// SIMATIC STEP 7 (V5.x) project Ciclo ppal
// program: Programa S7(2)
// program: TEST_DESBOBINADO
// program: TEST_CIZALLADO
// program: TEST_M_DESBOBINADO
// program: TEST_M_CIZALLADO
// program: TEST_G_DESBOBINADO
// program: TEST_G_CIZALLADO
// program: TEST_MODOS
// program: TEST_PESAJE
// program: TEST_GENERAL
// program: TEST_CORTAR
// program: TEST_ERRORES

SYMBOL_TABLE
"CONTADOR"	C 1	COUNTER	// Cuenta el numero de planchas cortadas
"Global"	DB 1	DB 1
"Modo1"	DB 2	DB 2
"Modo2"	DB 3	DB 3
"INFO_BOB"	DB 4	DB 4
"DESBOBINADO"	FB 1	FB 1	// Función que se encarga del desbobinado
"CIZALLADO"	FB 2	FB 2	// Funcion que se encaga del cizallado de planchas
"MULT_DESBOB"	FB 3	FB 3
"MULT_CIZA"	FB 4	FB 4
"GENERAL"	FB 5	FB 5
"MULT_GEN_DESB"	FB 6	FB 6
"MULT_GEN_CIZA"	FB 7	FB 7
"CORTA"	FB 8	FB 8
"MODO"	FB 9	FB 9
"ERRORES"	FC 1	FC 1
"PESAJE"	FC 2	FC 2	// Función de pesaje
"SCALE"	FC 105	FC 105	// Scaling Values
"BOBINA_COLOCADA"	I 124.0	BOOL
"S_SARTEN"	I 124.1	BOOL
"S_CACEROLA"	I 124.2	BOOL
"S_WOK"	I 124.3	BOOL
"S_PAELLERA"	I 124.4	BOOL
"PRESENCIA"	I 124.5	BOOL
"PALET"	I 124.6	BOOL
"SENSORARRIBA"	I 124.7	BOOL
"SENSORABAJO"	I 125.0	BOOL
"EXPULSADA"	I 125.1	BOOL
"ON"	I 125.2	BOOL
"BDT"	I 125.3	BOOL
"MODO_1"	I 125.4	BOOL
"MODO_2"	I 125.5	BOOL
"RESET"	I 125.6	BOOL
"SETA_PELIGROSA"	I 125.7	BOOL
"ERROR"	M 124.0	BOOL
"PESO_OUT"	MD 300	REAL
"CYCL_EXC"	OB 1	OB 1	// Cycle Execution
"MCENTRO"	PIW 651	INT
"IN_PESAJE"	PIW 653	INT
"ABRIRMCENTRO"	Q 100.0	BOOL
"CERRARMCENTRO"	Q 100.1	BOOL
"DESBOBINAR"	Q 100.2	BOOL
"EXPULSAR_BOBINA"	Q 100.3	BOOL
"EXPULSAR_PLANCHA"	Q 100.4	BOOL
"BAJAR_CUCHILLA"	Q 100.5	BOOL
"EXPULSAR_PALET"	Q 100.6	BOOL
"PRENSA"	Q 100.7	BOOL
"STBY_DESBOB"	Q 101.0	BOOL
"STBY_CIZA"	Q 101.1	BOOL
"TEMP_ERROR"	T 1	TIMER
END_SYMBOL_TABLE

FUNCTION_BLOCK "DESBOBINADO"	// FB 1
TITLE = DESBOBINADO
VERSION : 0.1
VAR_INPUT
  SENSOR : BOOL ;
  PRESENCIA : BOOL ;
  CENTRO : INT ;
  MCENTRO : INT ;
  Contador : COUNTER ;
  START : BOOL ;
  PLANCHAS : WORD  := W#16#100;
  ERROR : BOOL ;
  RESET : BOOL ;
END_VAR
VAR_OUTPUT
  ABRIRMCENTRO : BOOL ;
  DESBOBINAR : BOOL ;
  STBY : BOOL ;
END_VAR
VAR
  x31 : BOOL ;
  x32 : BOOL ;
  x33 : BOOL ;
  x34 : BOOL ;
  x30 : BOOL ;
  FP_PRESENCIA : BOOL ;
  BDT : BOOL ;
  FP_START : BOOL ;
  XERROR : BOOL ;
END_VAR
VAR_TEMP
  watchdog_master : BOOL ;
END_VAR
BEGIN
NETWORK
TITLE = Arranque
      SET;
      FP    #BDT;
      S     #x30;
      R     #x31;
      R     #x32;
      R     #x33;
      R     #x34;
NETWORK
TITLE =
      A     #RESET;
      R     #ABRIRMCENTRO;
      R     #DESBOBINAR;
      S     #x30;
      R     #x31;
      R     #x32;
      R     #x33;
      R     #x34;
      R     #XERROR;
NETWORK
TITLE =
      A     #ERROR;
      R     #ABRIRMCENTRO;
      R     #DESBOBINAR;
      R     #x30;
      R     #x31;
      R     #x32;
      R     #x33;
      R     #x34;
      S     #XERROR;
NETWORK
TITLE = x31 a x32
//Comparacion medida centro con medida nominal del centro para pasar de x31 a x32
      A     #x31;
      A(;
      L     #CENTRO;
      L     #MCENTRO;
      ==R;
      );
      R     #x31;
      S     #x32;
NETWORK
TITLE = x32 a x33
//Presencia detecta que la plancha esta en posicion para empezar el proceso de 
//desbobinado-cizallado
      A     #x32;
      A     #PRESENCIA;
      FP    #FP_PRESENCIA;
      R     #x32;
      S     #x33;
NETWORK
TITLE = x33 a x34
//Detecta que la plancha esta lista para ser cizallada
      A     #x33;
      A     #SENSOR;
      R     #x33;
      S     #x34;
NETWORK
TITLE = x34 a x33
//si el contador no ha acabado
      A     #x34;
      T     LD 1;
      TAK;
      T     LD 5;
      L     #Contador;
      T     LW 9;
      L     LD 5;
      L     LD 1;
      A     C [LW 9];
      AN    #SENSOR;
      R     #x34;
      S     #x33;
NETWORK
TITLE = x34 a X30
//si el contador ha cabado
      A     #x34;
      T     LD 1;
      TAK;
      T     LD 5;
      L     #Contador;
      T     LW 9;
      L     LD 5;
      L     LD 1;
      AN    C [LW 9];
      AN    #SENSOR;
      AN    #PRESENCIA;
      R     #x34;
      S     #x30;
NETWORK
TITLE = Tratamiento de bit de fin
      A     #x30;
      =     #STBY;
NETWORK
TITLE = Abrir centro
      A     #x31;
      =     #ABRIRMCENTRO;
NETWORK
TITLE = Carga del contador y desbobinado en x32
      A     #x32;
      S     #DESBOBINAR;
      L     #PLANCHAS;
      T     LD 1;
      TAK;
      T     LD 5;
      L     #Contador;
      T     LW 9;
      L     LD 5;
      L     LD 1;
      S     C [LW 9];
NETWORK
TITLE = Resta del contador y salida del x33
      A     #x33;
      S     #DESBOBINAR;
NETWORK
TITLE = Reset del desbobionado en x34
      A     #x34;
      R     #DESBOBINAR;
NETWORK
TITLE = De X30 a X31
      A     #START;
      FP    #FP_START;
      A     #x30;
      R     #x30;
      S     #x31;
END_FUNCTION_BLOCK

FUNCTION_BLOCK "CIZALLADO"	// FB 2
TITLE = CIZALLADO
VERSION : 0.1
VAR_INPUT
  SENSOR : BOOL ;
  SENSORABAJO : BOOL ;
  SENSORARRIBA : BOOL ;
  EXPULSADA : BOOL ;
  CONTADOR : COUNTER ;
  START : BOOL ;
  RESET : BOOL ;
  ERROR : BOOL ;
END_VAR
VAR_OUTPUT
  BAJARCUCHILLA : BOOL ;
  EXPULSARPLANCHA : BOOL ;
  STBY : BOOL ;
  BIT_OK : BOOL ;
END_VAR
VAR
  X41 : BOOL ;
  M3 : BOOL ;
  X43 : BOOL ;
  BDT : BOOL ;
  FP_START : BOOL ;
  INICORTAR : BOOL ;
  S2 : BOOL ;
  OK_CORTAR : BOOL ;
  STBY_CORTAR : BOOL ;
  CORTADO : BOOL ;
  XERROR : BOOL ;
  CORTAR : FB 8;
END_VAR
BEGIN
NETWORK
TITLE = Arranque
      SET;
      FP    #BDT;
      S     #X41;
      R     #M3;
      R     #X43;
      R     #INICORTAR;
      R     #CORTADO;
      R     #BIT_OK;
      R     #S2;
NETWORK
TITLE = De x41 a M3
      A     #X41;
      A     #SENSOR;
      A     #STBY_CORTAR;
      A     #START;
      FP    #FP_START;
      R     #X41;
      S     #M3;
NETWORK
TITLE = De M3 a x43
      A     #M3;
      A     #CORTADO;
      R     #M3;
      S     #X43;
NETWORK
TITLE = de x43 a x41
      A     #X43;
      A     #STBY_CORTAR;
      T     LD 0;
      TAK;
      T     LD 4;
      L     #CONTADOR;
      T     LW 8;
      L     LD 4;
      L     LD 0;
      AN    C [LW 8];
      R     #X43;
      S     #S2;
NETWORK
TITLE = de x43 a X41
      A     #X43;
      A     #STBY_CORTAR;
      T     LD 0;
      TAK;
      T     LD 4;
      L     #CONTADOR;
      T     LW 8;
      L     LD 4;
      L     LD 0;
      A     C [LW 8];
      R     #X43;
      S     #X41;
NETWORK
TITLE = Call M3
      CALL  #CORTAR (
           SENSORABAJO              := #SENSORABAJO,
           SENSORARRIBA             := #SENSORARRIBA,
           EXPULSADA                := #EXPULSADA,
           START                    := #INICORTAR,
           OK                       := #OK_CORTAR,
           ERROR                    := #ERROR,
           RESET                    := #RESET,
           BAJARCUCHILLA            := #BAJARCUCHILLA,
           EXPULSARPLANCHA          := #EXPULSARPLANCHA,
           BIT_OK                   := #CORTADO,
           STBY                     := #STBY_CORTAR);
NETWORK
TITLE = De M3 a X43
      A     #M3;
      A     #CORTADO;
      R     #M3;
      S     #X43;
NETWORK
TITLE = Salida M3
      A     #M3;
      =     #INICORTAR;
NETWORK
TITLE = Cuenta el numero de planchas cortadas
      A     #X43;
      =     #OK_CORTAR;
      T     LD 0;
      TAK;
      T     LD 4;
      L     #CONTADOR;
      T     LW 8;
      L     LD 4;
      L     LD 0;
      CD    C [LW 8];
NETWORK
TITLE = Salida X41
      A     #X41;
      =     #STBY;
NETWORK
TITLE = Salida S2
      A     #S2;
      =     #BIT_OK;
NETWORK
TITLE =
      A     #RESET;
      S     #X41;
      R     #M3;
      R     #X43;
      R     #INICORTAR;
      R     #CORTADO;
      R     #BIT_OK;
      R     #S2;
      R     #XERROR;
NETWORK
TITLE =
      A     #ERROR;
      R     #X41;
      R     #M3;
      R     #X43;
      R     #INICORTAR;
      R     #CORTADO;
      R     #BIT_OK;
      R     #S2;
      S     #XERROR;
END_FUNCTION_BLOCK

FUNCTION_BLOCK "MULT_DESBOB"	// FB 3
VERSION : 0.1
VAR_INPUT
  S_CACEROLA : BOOL ;
  S_SARTEN : BOOL ;
  S_PAELLERA : BOOL ;
  S_WOK : BOOL ;
  PRESENCIA : BOOL ;
  C_CACEROLA : INT ;
  C_SARTEN : INT ;
  C_WOK : INT ;
  C_PAELLERA : INT ;
  MCENTRO : INT ;
  CONTADOR : COUNTER ;
  PLANCHAS : WORD ;
  SARTEN : BOOL ;
  CACEROLA : BOOL ;
  WOK : BOOL ;
  PAELLERA : BOOL ;
  START : BOOL ;
  ERROR : BOOL ;
  RESET : BOOL ;
END_VAR
VAR_OUTPUT
  ABRIRMCENTRO : BOOL ;
  DESBOBINAR : BOOL ;
  BIT_OK : BOOL ;
  BIT_ERROR : BOOL ;
  STBY : BOOL ;
  STBY_SAR : BOOL ;
  STBY_CAC : BOOL ;
  STBY_WOK : BOOL ;
  STBY_PAELL : BOOL ;
END_VAR
VAR
  START_SAR : BOOL ;
  START_CAC : BOOL ;
  START_WOK : BOOL ;
  START_PAELL : BOOL ;
  FP_BDT : BOOL ;
  X1 : BOOL ;
  X2 : BOOL ;
  X3 : BOOL ;
  X4 : BOOL ;
  X5 : BOOL ;
  X6 : BOOL ;
  BDT : BOOL ;
  FP_START : BOOL ;
  FLAG_DESB : BOOL ;
  FP_DESBOB : BOOL ;
  F_START : BOOL ;
  FN_BDT : BOOL ;
  FN_X1 : BOOL ;
  SAR_DESBOB : FB 1;
  CAC_DESBOB : FB 1;
  WOK_DESBOB : FB 1;
  PAELL_DESBOB : FB 1;
END_VAR
BEGIN
NETWORK
TITLE = call del x2
      A     #X2;
      JCN   _001;
      S     #BDT;
      BLD   14;
      =     L 6.0;
      L     DINO;
      T     LW 4;
      CDB;
      OPN   DI [LW 4];
      TAR2  LD 0;
      A     DBX [AR2,P#0.1];
      =     #SAR_DESBOB.SENSOR;
      A     DBX [AR2,P#0.4];
      =     #SAR_DESBOB.PRESENCIA;
      L     DBW [AR2,P#4.0];
      T     #SAR_DESBOB.CENTRO;
      L     DBW [AR2,P#10.0];
      T     #SAR_DESBOB.MCENTRO;
      L     DBW [AR2,P#12.0];
      T     #SAR_DESBOB.Contador;
      A     DBX [AR2,P#20.0];
      =     #SAR_DESBOB.START;
      L     DBW [AR2,P#14.0];
      T     #SAR_DESBOB.PLANCHAS;
      A     DBX [AR2,P#16.5];
      =     #SAR_DESBOB.ERROR;
      A     DBX [AR2,P#16.6];
      =     #SAR_DESBOB.RESET;
      +AR2  P#24.0;
      UC    "DESBOBINADO";
      LAR2  LD 0;
      A     #SAR_DESBOB.ABRIRMCENTRO;
      =     DBX [AR2,P#18.0];
      A     #SAR_DESBOB.DESBOBINAR;
      =     DBX [AR2,P#18.1];
      A     #SAR_DESBOB.STBY;
      =     DBX [AR2,P#18.5];
      CDB;
      BLD   15;
_001: NOP   0;
NETWORK
TITLE = call del x3
      A     #X3;
      JCN   _002;
      S     #BDT;
      BLD   14;
      =     L 6.0;
      L     DINO;
      T     LW 4;
      CDB;
      OPN   DI [LW 4];
      TAR2  LD 0;
      A     DBX [AR2,P#0.0];
      =     #CAC_DESBOB.SENSOR;
      A     DBX [AR2,P#0.4];
      =     #CAC_DESBOB.PRESENCIA;
      L     DBW [AR2,P#2.0];
      T     #CAC_DESBOB.CENTRO;
      L     DBW [AR2,P#10.0];
      T     #CAC_DESBOB.MCENTRO;
      L     DBW [AR2,P#12.0];
      T     #CAC_DESBOB.Contador;
      A     DBX [AR2,P#20.1];
      =     #CAC_DESBOB.START;
      L     DBW [AR2,P#14.0];
      T     #CAC_DESBOB.PLANCHAS;
      A     DBX [AR2,P#16.5];
      =     #CAC_DESBOB.ERROR;
      A     DBX [AR2,P#16.6];
      =     #CAC_DESBOB.RESET;
      +AR2  P#42.0;
      UC    "DESBOBINADO";
      LAR2  LD 0;
      A     #CAC_DESBOB.ABRIRMCENTRO;
      =     DBX [AR2,P#18.0];
      A     #CAC_DESBOB.DESBOBINAR;
      =     DBX [AR2,P#18.1];
      A     #CAC_DESBOB.STBY;
      =     DBX [AR2,P#18.6];
      CDB;
      BLD   15;
_002: NOP   0;
NETWORK
TITLE = call del x4
      A     #X4;
      JCN   _003;
      S     #BDT;
      BLD   14;
      =     L 6.0;
      L     DINO;
      T     LW 4;
      CDB;
      OPN   DI [LW 4];
      TAR2  LD 0;
      A     DBX [AR2,P#0.3];
      =     #WOK_DESBOB.SENSOR;
      A     DBX [AR2,P#0.4];
      =     #WOK_DESBOB.PRESENCIA;
      L     DBW [AR2,P#6.0];
      T     #WOK_DESBOB.CENTRO;
      L     DBW [AR2,P#10.0];
      T     #WOK_DESBOB.MCENTRO;
      L     DBW [AR2,P#12.0];
      T     #WOK_DESBOB.Contador;
      A     DBX [AR2,P#20.2];
      =     #WOK_DESBOB.START;
      L     DBW [AR2,P#14.0];
      T     #WOK_DESBOB.PLANCHAS;
      A     DBX [AR2,P#16.5];
      =     #WOK_DESBOB.ERROR;
      A     DBX [AR2,P#16.6];
      =     #WOK_DESBOB.RESET;
      +AR2  P#60.0;
      UC    "DESBOBINADO";
      LAR2  LD 0;
      A     #WOK_DESBOB.ABRIRMCENTRO;
      =     DBX [AR2,P#18.0];
      A     #WOK_DESBOB.DESBOBINAR;
      =     DBX [AR2,P#18.1];
      A     #WOK_DESBOB.STBY;
      =     DBX [AR2,P#18.7];
      CDB;
      BLD   15;
_003: NOP   0;
NETWORK
TITLE = call del x5
      A     #X5;
      JCN   _004;
      S     #BDT;
      BLD   14;
      =     L 6.0;
      L     DINO;
      T     LW 4;
      CDB;
      OPN   DI [LW 4];
      TAR2  LD 0;
      A     DBX [AR2,P#0.2];
      =     #PAELL_DESBOB.SENSOR;
      A     DBX [AR2,P#0.4];
      =     #PAELL_DESBOB.PRESENCIA;
      L     DBW [AR2,P#8.0];
      T     #PAELL_DESBOB.CENTRO;
      L     DBW [AR2,P#10.0];
      T     #PAELL_DESBOB.MCENTRO;
      L     DBW [AR2,P#12.0];
      T     #PAELL_DESBOB.Contador;
      A     DBX [AR2,P#20.3];
      =     #PAELL_DESBOB.START;
      L     DBW [AR2,P#14.0];
      T     #PAELL_DESBOB.PLANCHAS;
      A     DBX [AR2,P#16.5];
      =     #PAELL_DESBOB.ERROR;
      A     DBX [AR2,P#16.6];
      =     #PAELL_DESBOB.RESET;
      +AR2  P#78.0;
      UC    "DESBOBINADO";
      LAR2  LD 0;
      A     #PAELL_DESBOB.ABRIRMCENTRO;
      =     DBX [AR2,P#18.0];
      A     #PAELL_DESBOB.DESBOBINAR;
      =     DBX [AR2,P#18.1];
      A     #PAELL_DESBOB.STBY;
      =     DBX [AR2,P#18.4];
      CDB;
      BLD   15;
_004: NOP   0;
NETWORK
TITLE = salida x2
      A     #X2;
      =     #START_SAR;
NETWORK
TITLE = salida x3
      A     #X3;
      =     #START_CAC;
NETWORK
TITLE = salida x4
      A     #X4;
      =     #START_WOK;
NETWORK
TITLE = salida x5
      A     #X5;
      =     #START_PAELL;
NETWORK
TITLE = Arranque
      SET;
      FP    #FP_BDT;
      R     #START_SAR;
      R     #START_CAC;
      R     #START_WOK;
      R     #START_PAELL;
      S     #X1;
      R     #X2;
      R     #X3;
      R     #X4;
      R     #X5;
      R     #X6;
NETWORK
TITLE = guardado de flanco de start
      A     #START;
      FP    #FP_START;
      =     #F_START;
NETWORK
TITLE = de x1 x2
      A     #F_START;
      A     #X1;
      A     #SARTEN;
      R     #X1;
      S     #X2;
NETWORK
TITLE = de x1 a x3
      A     #F_START;
      A     #X1;
      A     #CACEROLA;
      R     #X1;
      S     #X3;
NETWORK
TITLE = de x1 a x4
      A     #F_START;
      A     #X1;
      A     #WOK;
      R     #X1;
      S     #X4;
NETWORK
TITLE = de x1 a x5
      A     #F_START;
      A     #X1;
      A     #PAELLERA;
      R     #X1;
      S     #X5;
NETWORK
TITLE = Guardado flag desbobinado
      A     #DESBOBINAR;
      FP    #FP_DESBOB;
      S     #FLAG_DESB;
NETWORK
TITLE = de x2 a x6
      A     #X2;
      A     #FLAG_DESB;
      A     #STBY_SAR;
      R     #FLAG_DESB;
      R     #X2;
      S     #X6;
NETWORK
TITLE = de x3 a x6
      A     #X3;
      A     #FLAG_DESB;
      A     #STBY_CAC;
      R     #FLAG_DESB;
      R     #X3;
      S     #X6;
NETWORK
TITLE = de x4 a x6
      A     #X4;
      A     #FLAG_DESB;
      A     #STBY_WOK;
      R     #FLAG_DESB;
      R     #X4;
      S     #X6;
NETWORK
TITLE = de x5 a x6
      A     #X5;
      A     #FLAG_DESB;
      A     #STBY_PAELL;
      R     #FLAG_DESB;
      R     #X5;
      S     #X6;
NETWORK
TITLE = salida x1
      A     #X1;
      =     #STBY;
NETWORK
TITLE = salida x6 
      A     #X6;
      =     #BIT_OK;
NETWORK
TITLE = error, sin prgramar
      A     #RESET;
      A(;
      A(;
      O(;
      A     #STBY_CAC;
      A     #X3;
      );
      O(;
      A     #STBY_SAR;
      A     #X2;
      );
      O(;
      A     #STBY_WOK;
      A     #X4;
      );
      O(;
      A     #STBY_PAELL;
      A     #X5;
      );
      );
      O     #X6;
      );
      R     #BDT;
      R     #BIT_OK;
      R     #BIT_ERROR;
      S     #X1;
      R     #X2;
      R     #X3;
      R     #X4;
      R     #X5;
      R     #X6;
      R     #START_SAR;
      R     #START_CAC;
      R     #START_WOK;
      R     #START_PAELL;
      R     #FLAG_DESB;
      R     #ABRIRMCENTRO;
      R     #DESBOBINAR;
END_FUNCTION_BLOCK

FUNCTION_BLOCK "MULT_CIZA"	// FB 4
VERSION : 0.1
VAR_INPUT
  S_CACEROLA : BOOL ;
  S_WOK : BOOL ;
  S_SARTEN : BOOL ;
  S_PAELLERA : BOOL ;
  SENSORARRIBA : BOOL ;
  SENSORABAJO : BOOL ;
  EXPULSADA : BOOL ;
  CONTADOR : COUNTER ;
  SARTEN : BOOL ;
  CACEROLA : BOOL ;
  WOK : BOOL ;
  PAELLERA : BOOL ;
  START : BOOL ;
  ERROR : BOOL ;
  RESET : BOOL ;
END_VAR
VAR_OUTPUT
  EXPULSARPLANCHA : BOOL ;
  BAJARCUCHILLA : BOOL ;
  BIT_OK : BOOL ;
  STBY : BOOL ;
END_VAR
VAR
  START_SAR : BOOL ;
  START_CAC : BOOL ;
  START_WOK : BOOL ;
  START_PAELL : BOOL ;
  X1 : BOOL ;
  X2 : BOOL ;
  X3 : BOOL ;
  X4 : BOOL ;
  X5 : BOOL ;
  FP_START : BOOL ;
  F_START : BOOL ;
  STBY_SAR : BOOL ;
  STBY_CAC : BOOL ;
  STBY_WOK : BOOL ;
  STBY_PAELL : BOOL ;
  OK : BOOL ;
  BDT : BOOL ;
  X6 : BOOL ;
  RESET_CIZA : BOOL ;
  FP_RESET : BOOL ;
  CAC_CIZA : FB 2;
  SAR_CIZA : FB 2;
  WOK_CIZA : FB 2;
  PAELL_CIZA : FB 2;
END_VAR
BEGIN
NETWORK
TITLE = Arranque
      SET;
      FP    #BDT;
      S     #X1;
      R     #X2;
      R     #X3;
      R     #X4;
      R     #X5;
      R     #X6;
NETWORK
TITLE = De x1 a x2
      A     #START;
      A     #SARTEN;
      A     #X1;
      R     #X1;
      S     #X2;
NETWORK
TITLE = de x1 a x3
      A     #START;
      A     #CACEROLA;
      A     #X1;
      R     #X1;
      S     #X3;
NETWORK
TITLE = de x1 a x4
      A     #START;
      A     #WOK;
      A     #X1;
      R     #X1;
      S     #X4;
NETWORK
TITLE = de x1 a x5
      A     #START;
      A     #PAELLERA;
      A     #X1;
      R     #X1;
      S     #X5;
NETWORK
TITLE = de x2-5 a x1
      A     #OK;
      A(;
      O     #X2;
      O     #X3;
      O     #X4;
      O     #X5;
      );
      R     #X2;
      R     #X3;
      R     #X4;
      R     #X5;
      S     #X1;
NETWORK
TITLE = call del x2
      A     #X2;
      JCN   _001;
      BLD   14;
      =     L 6.0;
      L     DINO;
      T     LW 4;
      CDB;
      OPN   DI [LW 4];
      TAR2  LD 0;
      A     DBX [AR2,P#0.2];
      =     #SAR_CIZA.SENSOR;
      A     DBX [AR2,P#0.5];
      =     #SAR_CIZA.SENSORABAJO;
      A     DBX [AR2,P#0.4];
      =     #SAR_CIZA.SENSORARRIBA;
      A     DBX [AR2,P#0.6];
      =     #SAR_CIZA.EXPULSADA;
      L     DBW [AR2,P#2.0];
      T     #SAR_CIZA.CONTADOR;
      A     DBX [AR2,P#8.0];
      =     #SAR_CIZA.START;
      A     DBX [AR2,P#10.2];
      =     #SAR_CIZA.RESET;
      A     DBX [AR2,P#4.5];
      =     #SAR_CIZA.ERROR;
      +AR2  P#28.0;
      UC    "CIZALLADO";
      LAR2  LD 0;
      A     #SAR_CIZA.BAJARCUCHILLA;
      =     DBX [AR2,P#6.1];
      A     #SAR_CIZA.EXPULSARPLANCHA;
      =     DBX [AR2,P#6.0];
      A     #SAR_CIZA.STBY;
      =     DBX [AR2,P#9.3];
      A     #SAR_CIZA.BIT_OK;
      =     DBX [AR2,P#9.7];
      CDB;
      BLD   15;
_001: NOP   0;
NETWORK
TITLE = call del x3
      A     #X3;
      JCN   _002;
      BLD   14;
      =     L 6.0;
      L     DINO;
      T     LW 4;
      CDB;
      OPN   DI [LW 4];
      TAR2  LD 0;
      A     DBX [AR2,P#0.0];
      =     #CAC_CIZA.SENSOR;
      A     DBX [AR2,P#0.5];
      =     #CAC_CIZA.SENSORABAJO;
      A     DBX [AR2,P#0.4];
      =     #CAC_CIZA.SENSORARRIBA;
      A     DBX [AR2,P#0.6];
      =     #CAC_CIZA.EXPULSADA;
      L     DBW [AR2,P#2.0];
      T     #CAC_CIZA.CONTADOR;
      A     DBX [AR2,P#8.1];
      =     #CAC_CIZA.START;
      A     DBX [AR2,P#10.2];
      =     #CAC_CIZA.RESET;
      A     DBX [AR2,P#4.5];
      =     #CAC_CIZA.ERROR;
      +AR2  P#12.0;
      UC    "CIZALLADO";
      LAR2  LD 0;
      A     #CAC_CIZA.BAJARCUCHILLA;
      =     DBX [AR2,P#6.1];
      A     #CAC_CIZA.EXPULSARPLANCHA;
      =     DBX [AR2,P#6.0];
      A     #CAC_CIZA.STBY;
      =     DBX [AR2,P#9.4];
      A     #CAC_CIZA.BIT_OK;
      =     DBX [AR2,P#9.7];
      CDB;
      BLD   15;
_002: NOP   0;
NETWORK
TITLE = call del x4
      A     #X4;
      JCN   _003;
      BLD   14;
      =     L 6.0;
      L     DINO;
      T     LW 4;
      CDB;
      OPN   DI [LW 4];
      TAR2  LD 0;
      A     DBX [AR2,P#0.1];
      =     #WOK_CIZA.SENSOR;
      A     DBX [AR2,P#0.5];
      =     #WOK_CIZA.SENSORABAJO;
      A     DBX [AR2,P#0.4];
      =     #WOK_CIZA.SENSORARRIBA;
      A     DBX [AR2,P#0.6];
      =     #WOK_CIZA.EXPULSADA;
      L     DBW [AR2,P#2.0];
      T     #WOK_CIZA.CONTADOR;
      A     DBX [AR2,P#8.2];
      =     #WOK_CIZA.START;
      A     DBX [AR2,P#10.2];
      =     #WOK_CIZA.RESET;
      A     DBX [AR2,P#4.5];
      =     #WOK_CIZA.ERROR;
      +AR2  P#44.0;
      UC    "CIZALLADO";
      LAR2  LD 0;
      A     #WOK_CIZA.BAJARCUCHILLA;
      =     DBX [AR2,P#6.1];
      A     #WOK_CIZA.EXPULSARPLANCHA;
      =     DBX [AR2,P#6.0];
      A     #WOK_CIZA.STBY;
      =     DBX [AR2,P#9.5];
      A     #WOK_CIZA.BIT_OK;
      =     DBX [AR2,P#9.7];
      CDB;
      BLD   15;
_003: NOP   0;
NETWORK
TITLE = call del x5
      A     #X5;
      JCN   _004;
      BLD   14;
      =     L 6.0;
      L     DINO;
      T     LW 4;
      CDB;
      OPN   DI [LW 4];
      TAR2  LD 0;
      A     DBX [AR2,P#0.3];
      =     #PAELL_CIZA.SENSOR;
      A     DBX [AR2,P#0.5];
      =     #PAELL_CIZA.SENSORABAJO;
      A     DBX [AR2,P#0.4];
      =     #PAELL_CIZA.SENSORARRIBA;
      A     DBX [AR2,P#0.6];
      =     #PAELL_CIZA.EXPULSADA;
      L     DBW [AR2,P#2.0];
      T     #PAELL_CIZA.CONTADOR;
      A     DBX [AR2,P#8.3];
      =     #PAELL_CIZA.START;
      A     DBX [AR2,P#10.2];
      =     #PAELL_CIZA.RESET;
      A     DBX [AR2,P#4.5];
      =     #PAELL_CIZA.ERROR;
      +AR2  P#60.0;
      UC    "CIZALLADO";
      LAR2  LD 0;
      A     #PAELL_CIZA.BAJARCUCHILLA;
      =     DBX [AR2,P#6.1];
      A     #PAELL_CIZA.EXPULSARPLANCHA;
      =     DBX [AR2,P#6.0];
      A     #PAELL_CIZA.STBY;
      =     DBX [AR2,P#9.6];
      A     #PAELL_CIZA.BIT_OK;
      =     DBX [AR2,P#9.7];
      CDB;
      BLD   15;
_004: NOP   0;
NETWORK
TITLE = salida x2
      A     #X2;
      =     #START_SAR;
NETWORK
TITLE = salida x3
      A     #X3;
      =     #START_CAC;
NETWORK
TITLE = salida x4
      A     #X4;
      =     #START_WOK;
NETWORK
TITLE = salida x5
      A     #X5;
      =     #START_PAELL;
NETWORK
TITLE =
      A     #X1;
      =     #STBY;
NETWORK
TITLE =
      A(;
      O     #X2;
      O     #X3;
      O     #X4;
      O     #X5;
      );
      FP    #FP_RESET;
      =     #RESET_CIZA;
NETWORK
TITLE =
      A     #RESET;
      A(;
      A(;
      O(;
      A     #STBY_CAC;
      A     #X3;
      );
      O(;
      A     #STBY_SAR;
      A     #X2;
      );
      O(;
      A     #STBY_WOK;
      A     #X4;
      );
      O(;
      A     #STBY_PAELL;
      A     #X5;
      );
      );
      O     #X6;
      );
      S     #X1;
      R     #X2;
      R     #X3;
      R     #X4;
      R     #X5;
      R     #EXPULSARPLANCHA;
      R     #BAJARCUCHILLA;
      R     #BIT_OK;
END_FUNCTION_BLOCK

FUNCTION_BLOCK "GENERAL"	// FB 5
VERSION : 0.1
VAR_INPUT
  BOBINA_COLOCADA : BOOL ;
  MCENTRO : INT ;
  IN_PESAJE : INT ;
  S_SARTEN : BOOL ;
  S_CACEROLA : BOOL ;
  S_WOK : BOOL ;
  S_PAELLERA : BOOL ;
  PRESENCIA : BOOL ;
  CONTADOR : COUNTER ;
  PALET : BOOL ;
  SENSORARRIBA : BOOL ;
  SENSORABAJO : BOOL ;
  EXPULSADA : BOOL ;
  ON : BOOL ;
  MODO_1 : BOOL ;
  MODO_2 : BOOL ;
  ERROR : BOOL ;
  RESET : BOOL ;
END_VAR
VAR_OUTPUT
  PESO_OUT : REAL ;
  ABRIRMCENTRO : BOOL ;
  CERRARMCENTRO : BOOL ;
  DESBOBINAR : BOOL ;
  EXPULSAR_BOBINA : BOOL ;
  EXPULSAR_PLANCHA : BOOL ;
  BAJAR_CUCHILLA : BOOL ;
  EXPULSAR_PALET : BOOL ;
  PRENSA : BOOL ;
  STBY_DESBOB_1 : BOOL ;
  STBY_CIZA_1 : BOOL ;
END_VAR
VAR
  SARTEN : BOOL ;
  CACEROLA : BOOL ;
  WOK : BOOL ;
  PAELLERA : BOOL ;
  START : BOOL ;
  BDT : BOOL ;
  STBY_DESBOB : BOOL ;
  STBY_CIZA : BOOL ;
  X0 : BOOL ;
  X1 : BOOL ;
  FP_ON : BOOL ;
  FP_STBY : BOOL ;
  FP_BDT : BOOL ;
  MODOS : FB 9;
  STBY_MODOS : BOOL ;
  DESBOB : FB 6;
  CIZA : FB 7;
END_VAR
BEGIN
NETWORK
TITLE = CALL DEL CIZALLADO
      SET;
      BLD   14;
      =     L 6.0;
      L     DINO;
      T     LW 4;
      CDB;
      OPN   DI [LW 4];
      TAR2  LD 0;
      A     DBX [AR2,P#18.4];
      =     #CIZA.START;
      A     DBX [AR2,P#6.0];
      =     #CIZA.S_SARTEN;
      A     DBX [AR2,P#6.1];
      =     #CIZA.S_CACEROLA;
      A     DBX [AR2,P#6.2];
      =     #CIZA.S_WOK;
      A     DBX [AR2,P#6.3];
      =     #CIZA.S_PAELLERA;
      L     DBW [AR2,P#8.0];
      T     #CIZA.CONTADOR;
      A     DBX [AR2,P#10.0];
      =     #CIZA.PALET;
      A     DBX [AR2,P#10.1];
      =     #CIZA.SENSORARRIBA;
      A     DBX [AR2,P#10.2];
      =     #CIZA.SENSORABAJO;
      A     DBX [AR2,P#10.3];
      =     #CIZA.EXPULSADA;
      A     DBX [AR2,P#18.0];
      =     #CIZA.SARTEN;
      A     DBX [AR2,P#18.1];
      =     #CIZA.CACEROLA;
      A     DBX [AR2,P#18.2];
      =     #CIZA.WOK;
      A     DBX [AR2,P#18.3];
      =     #CIZA.PAELLERA;
      A     DBX [AR2,P#10.7];
      =     #CIZA.ERROR;
      A     DBX [AR2,P#11.0];
      =     #CIZA.RESET;
      +AR2  P#150.0;
      UC    "MULT_GEN_CIZA";
      LAR2  LD 0;
      A     #CIZA.EXPULSAR_PLANCHA;
      =     DBX [AR2,P#16.4];
      A     #CIZA.BAJAR_CUCHILLA;
      =     DBX [AR2,P#16.5];
      A     #CIZA.EXPULSAR_PALET;
      =     DBX [AR2,P#16.6];
      A     #CIZA.STBY;
      =     DBX [AR2,P#18.7];
      CDB;
      BLD   15;
NETWORK
TITLE = CALL DEL DESBOBINADO
      SET;
      BLD   14;
      =     L 6.0;
      L     DINO;
      T     LW 4;
      CDB;
      OPN   DI [LW 4];
      TAR2  LD 0;
      A     DBX [AR2,P#18.4];
      =     #DESBOB.START;
      A     DBX [AR2,P#0.0];
      =     #DESBOB.BOBINA_COLOCADA;
      L     DBW [AR2,P#2.0];
      T     #DESBOB.MCENTRO;
      L     DBW [AR2,P#4.0];
      T     #DESBOB.IN_PESAJE;
      A     DBX [AR2,P#6.0];
      =     #DESBOB.S_SARTEN;
      A     DBX [AR2,P#6.1];
      =     #DESBOB.S_CACEROLA;
      A     DBX [AR2,P#6.2];
      =     #DESBOB.S_WOK;
      A     DBX [AR2,P#6.3];
      =     #DESBOB.S_PAELLERA;
      A     DBX [AR2,P#6.4];
      =     #DESBOB.PRESENCIA;
      L     DBW [AR2,P#8.0];
      T     #DESBOB.CONTADOR;
      A     DBX [AR2,P#10.7];
      =     #DESBOB.ERROR;
      A     DBX [AR2,P#11.0];
      =     #DESBOB.RESET;
      A     DBX [AR2,P#18.0];
      =     #DESBOB.SARTEN;
      A     DBX [AR2,P#18.1];
      =     #DESBOB.CACEROLA;
      A     DBX [AR2,P#18.2];
      =     #DESBOB.WOK;
      A     DBX [AR2,P#18.3];
      =     #DESBOB.PAELLERA;
      +AR2  P#28.0;
      UC    "MULT_GEN_DESB";
      LAR2  LD 0;
      L     #DESBOB.PESO_OUT;
      T     DBD [AR2,P#12.0];
      A     #DESBOB.ABRIRMCENTRO;
      =     DBX [AR2,P#16.0];
      A     #DESBOB.CERRARMCENTRO;
      =     DBX [AR2,P#16.1];
      A     #DESBOB.DESBOBINAR;
      =     DBX [AR2,P#16.2];
      A     #DESBOB.EXPULSAR_BOBINA;
      =     DBX [AR2,P#16.3];
      A     #DESBOB.STBY;
      =     DBX [AR2,P#18.6];
      A     #DESBOB.SARTEN;
      =     DBX [AR2,P#18.0];
      A     #DESBOB.CACEROLA;
      =     DBX [AR2,P#18.1];
      A     #DESBOB.WOK;
      =     DBX [AR2,P#18.2];
      A     #DESBOB.PAELLERA;
      =     DBX [AR2,P#18.3];
      CDB;
      BLD   15;
NETWORK
TITLE =
      CALL  #MODOS (
           MODO1                    := #MODO_1,
           MODO2                    := #MODO_2,
           STBY                     := #STBY_MODOS);
NETWORK
TITLE = DE X0 A X1
      A     #ON;
      FP    #FP_ON;
      A     #X0;
      AN    #STBY_MODOS;
      R     #X0;
      S     #X1;
NETWORK
TITLE = ARRANQUE
      SET;
      FP    #FP_BDT;
      =     #BDT;
      S     #X0;
      R     #X1;
NETWORK
TITLE = DE X1 A X0
      A(;
      A     #STBY_CIZA;
      A     #STBY_DESBOB;
      );
      FP    #FP_STBY;
      R     #X1;
      S     #X0;
NETWORK
TITLE = SALIDA DE X1
      A     #X1;
      =     #START;
NETWORK
TITLE = MANEJO DE LA PRENSA
      A     #DESBOBINAR;
      =     #PRENSA;
NETWORK
TITLE = VARIOS
      A     #STBY_DESBOB;
      =     #STBY_DESBOB_1;
      A     #STBY_CIZA;
      =     #STBY_CIZA_1;
NETWORK
TITLE =
      A     #RESET;
      R     #X1;
      S     #X0;
END_FUNCTION_BLOCK

FUNCTION_BLOCK "MULT_GEN_DESB"	// FB 6
VERSION : 0.1
VAR_INPUT
  START : BOOL ;
  BOBINA_COLOCADA : BOOL ;
  MCENTRO : INT ;
  IN_PESAJE : INT ;
  S_SARTEN : BOOL ;
  S_CACEROLA : BOOL ;
  S_WOK : BOOL ;
  S_PAELLERA : BOOL ;
  PRESENCIA : BOOL ;
  CONTADOR : COUNTER ;
  ERROR : BOOL ;
  RESET : BOOL ;
END_VAR
VAR_OUTPUT
  PESO_OUT : REAL ;
  ABRIRMCENTRO : BOOL ;
  CERRARMCENTRO : BOOL ;
  DESBOBINAR : BOOL ;
  EXPULSAR_BOBINA : BOOL ;
  STBY : BOOL ;
END_VAR
VAR_IN_OUT
  SARTEN : BOOL ;
  CACEROLA : BOOL ;
  WOK : BOOL ;
  PAELLERA : BOOL ;
END_VAR
VAR
  X0 : BOOL ;
  X1 : BOOL ;
  X2 : BOOL ;
  X3 : BOOL ;
  X4 : BOOL ;
  X5 : BOOL ;
  FP_START : BOOL ;
  BDT_PESAJE : BOOL ;
  RECIBIDO_PESAJE : BOOL ;
  START_PESAJE : BOOL ;
  STBY_PESAJE : BOOL ;
  OK_DESBOB : BOOL ;
  START_DESBOB : BOOL ;
  OK_DESBOB_1 : BOOL ;
  STBY_DESBOB : BOOL ;
  FP_OK_DESBOB : BOOL ;
  BDT : BOOL ;
  FN_BDT : BOOL ;
  DESBOB : FB 3;
  XERROR : BOOL ;
END_VAR
BEGIN
NETWORK
TITLE = DE X1 A X2
      A     #X1;
      A     #BOBINA_COLOCADA;
      R     #X1;
      S     #X2;
NETWORK
TITLE = DE X0 A X1
      A     #START;
      FP    #FP_START;
      A     #X0;
      R     #X0;
      S     #X1;
NETWORK
TITLE = ARRANQUE
      SET;
      FP    #BDT;
      R     #BDT_PESAJE;
      R     #START_PESAJE;
      R     #START_DESBOB;
      S     #X0;
      R     #X1;
      R     #X2;
      R     #X3;
      R     #X4;
      R     #X5;
      R     #XERROR;
NETWORK
TITLE = ERROR, NO PROGRAMADO
      A     #RESET;
      R     #BDT_PESAJE;
      R     #START_PESAJE;
      R     #START_DESBOB;
      S     #X0;
      R     #X1;
      R     #X2;
      R     #X3;
      R     #X4;
      R     #X5;
      R     #XERROR;
NETWORK
TITLE = CALL DESBOBINADOR
      SET;
      BLD   14;
      =     L 6.0;
      L     DINO;
      T     LW 4;
      CDB;
      OPN   DI [LW 4];
      TAR2  LD 0;
      A     DBX [AR2,P#6.1];
      =     #DESBOB.S_CACEROLA;
      A     DBX [AR2,P#6.0];
      =     #DESBOB.S_SARTEN;
      A     DBX [AR2,P#6.3];
      =     #DESBOB.S_PAELLERA;
      A     DBX [AR2,P#6.2];
      =     #DESBOB.S_WOK;
      A     DBX [AR2,P#6.4];
      =     #DESBOB.PRESENCIA;
      OPN   DI 4;
      L     DIW 0;
      OPN   DI [LW 4];
      T     #DESBOB.C_CACEROLA;
      OPN   DI 4;
      L     DIW 2;
      OPN   DI [LW 4];
      T     #DESBOB.C_SARTEN;
      OPN   DI 4;
      L     DIW 4;
      OPN   DI [LW 4];
      T     #DESBOB.C_WOK;
      OPN   DI 4;
      L     DIW 6;
      OPN   DI [LW 4];
      T     #DESBOB.C_PAELLERA;
      L     DBW [AR2,P#2.0];
      T     #DESBOB.MCENTRO;
      L     DBW [AR2,P#8.0];
      T     #DESBOB.CONTADOR;
      OPN   DI 1;
      L     DIW 16;
      OPN   DI [LW 4];
      T     #DESBOB.PLANCHAS;
      A     DBX [AR2,P#18.0];
      =     #DESBOB.SARTEN;
      A     DBX [AR2,P#18.1];
      =     #DESBOB.CACEROLA;
      A     DBX [AR2,P#18.2];
      =     #DESBOB.WOK;
      A     DBX [AR2,P#18.3];
      =     #DESBOB.PAELLERA;
      A     DBX [AR2,P#0.0];
      =     #DESBOB.START;
      A     DBX [AR2,P#10.0];
      =     #DESBOB.ERROR;
      A     DBX [AR2,P#10.1];
      =     #DESBOB.RESET;
      +AR2  P#24.0;
      UC    "MULT_DESBOB";
      LAR2  LD 0;
      A     #DESBOB.ABRIRMCENTRO;
      =     DBX [AR2,P#16.0];
      A     #DESBOB.DESBOBINAR;
      =     DBX [AR2,P#16.2];
      A     #DESBOB.BIT_OK;
      =     DBX [AR2,P#21.3];
      A     #DESBOB.STBY;
      =     DBX [AR2,P#21.6];
      CDB;
      BLD   15;
NETWORK
TITLE = DE X2 A X3
      A     #X2;
      A(;
      O     #SARTEN;
      O     #CACEROLA;
      O     #WOK;
      O     #PAELLERA;
      );
      R     #X2;
      S     #X3;
NETWORK
TITLE = DE X3 A X4
      A     #OK_DESBOB;
      FP    #FP_OK_DESBOB;
      A     #X3;
      R     #X3;
      R     #OK_DESBOB;
      S     #X4;
NETWORK
TITLE = DE X4 A X5
      A     #X4;
      A(;
      L     #MCENTRO;
      L     0;
      ==I;
      );
      R     #X4;
      S     #X5;
NETWORK
TITLE = DE X5 A X0
      A     #X5;
      AN    #BOBINA_COLOCADA;
      R     #X5;
      S     #X0;
NETWORK
TITLE = CALL PESAJE
      SET;
      CALL  "PESAJE" (
           in                       := #IN_PESAJE,
           PESO_SARTEN              := "Global".PESO_SARTEN,
           PESO_CACEROLA            := "Global".PESO_CACEROLA,
           PESO_WOK                 := "Global".PESO_WOK,
           PESO_PAELLERA            := "Global".PESO_PAELLERA,
           bit_de_trabajo           := #BDT_PESAJE,
           RECIBIDO                 := #RECIBIDO_PESAJE,
           START                    := #START_PESAJE,
           stby                     := #STBY_PESAJE,
           SARTEN                   := #SARTEN,
           CACEROLA                 := #CACEROLA,
           WOK                      := #WOK,
           PAELLERA                 := #PAELLERA,
           PESO_OUT                 := #PESO_OUT);
NETWORK
TITLE =
      A     #ERROR;
      R     #BDT_PESAJE;
      R     #START_PESAJE;
      R     #START_DESBOB;
      R     #X0;
      R     #X1;
      R     #X2;
      R     #X3;
      R     #X4;
      R     #X5;
      S     #XERROR;
NETWORK
TITLE = SALIDA X2
      A     #X2;
      =     #START_PESAJE;
NETWORK
TITLE = SALIDA X3
      A     #X3;
      =     #START_DESBOB;
      R     #BDT_PESAJE;
NETWORK
TITLE = SALIDA X4
      A     #X4;
      =     #CERRARMCENTRO;
NETWORK
TITLE = SALIDA X5
      A     #X5;
      =     #EXPULSAR_BOBINA;
NETWORK
TITLE = SALIDA X0
      A     #X0;
      =     #STBY;
NETWORK
TITLE = RESET BDT PESAJE EN X1
      A     #X1;
      S     #BDT_PESAJE;
END_FUNCTION_BLOCK

FUNCTION_BLOCK "MULT_GEN_CIZA"	// FB 7
VERSION : 0.1
VAR_INPUT
  START : BOOL ;
  S_SARTEN : BOOL ;
  S_CACEROLA : BOOL ;
  S_WOK : BOOL ;
  S_PAELLERA : BOOL ;
  CONTADOR : COUNTER ;
  PALET : BOOL ;
  SENSORARRIBA : BOOL ;
  SENSORABAJO : BOOL ;
  EXPULSADA : BOOL ;
  SARTEN : BOOL ;
  CACEROLA : BOOL ;
  WOK : BOOL ;
  PAELLERA : BOOL ;
  ERROR : BOOL ;
  RESET : BOOL ;
END_VAR
VAR_OUTPUT
  EXPULSAR_PLANCHA : BOOL ;
  BAJAR_CUCHILLA : BOOL ;
  EXPULSAR_PALET : BOOL ;
  STBY : BOOL ;
END_VAR
VAR
  X10 : BOOL ;
  X11 : BOOL ;
  X12 : BOOL ;
  BDT : BOOL ;
  START_CIZA : BOOL ;
  STBY_CIZA : BOOL ;
  FP_STBY_CIZA : BOOL ;
  X0 : BOOL ;
  FP_START : BOOL ;
  FP : BOOL ;
  XERROR : BOOL ;
  CIZA : FB 4;
END_VAR
BEGIN
NETWORK
TITLE = Arranque
      SET;
      FP    #BDT;
      S     #X0;
      R     #X10;
      R     #X11;
      R     #X12;
NETWORK
TITLE = de x0 a x10
      A     #START;
      FP    #FP_START;
      A     #X0;
      R     #X0;
      S     #X10;
NETWORK
TITLE = de x10 a x11
      A     #X10;
      A(;
      O     #SARTEN;
      O     #CACEROLA;
      O     #WOK;
      O     #PAELLERA;
      );
      A     #PALET;
      R     #X10;
      S     #X11;
NETWORK
TITLE = de x11 a x12
      A     #STBY_CIZA;
      FP    #FP_STBY_CIZA;
      A     #X11;
      R     #X11;
      S     #X12;
NETWORK
TITLE = de x12 a x0
      A     #X12;
      AN    #PALET;
      R     #X12;
      S     #X0;
NETWORK
TITLE = call cizado
      BLD   14;
      =     L 6.0;
      L     DINO;
      T     LW 4;
      CDB;
      OPN   DI [LW 4];
      TAR2  LD 0;
      A     DBX [AR2,P#0.2];
      =     #CIZA.S_CACEROLA;
      A     DBX [AR2,P#0.3];
      =     #CIZA.S_WOK;
      A     DBX [AR2,P#0.1];
      =     #CIZA.S_SARTEN;
      A     DBX [AR2,P#0.4];
      =     #CIZA.S_PAELLERA;
      A     DBX [AR2,P#4.1];
      =     #CIZA.SENSORARRIBA;
      A     DBX [AR2,P#4.2];
      =     #CIZA.SENSORABAJO;
      A     DBX [AR2,P#4.3];
      =     #CIZA.EXPULSADA;
      L     DBW [AR2,P#2.0];
      T     #CIZA.CONTADOR;
      A     DBX [AR2,P#4.4];
      =     #CIZA.SARTEN;
      A     DBX [AR2,P#4.5];
      =     #CIZA.CACEROLA;
      A     DBX [AR2,P#4.6];
      =     #CIZA.WOK;
      A     DBX [AR2,P#4.7];
      =     #CIZA.PAELLERA;
      A     DBX [AR2,P#0.0];
      =     #CIZA.START;
      A     DBX [AR2,P#5.0];
      =     #CIZA.ERROR;
      A     DBX [AR2,P#5.1];
      =     #CIZA.RESET;
      +AR2  P#10.0;
      UC    "MULT_CIZA";
      LAR2  LD 0;
      A     #CIZA.EXPULSARPLANCHA;
      =     DBX [AR2,P#6.0];
      A     #CIZA.BAJARCUCHILLA;
      =     DBX [AR2,P#6.1];
      A     #CIZA.STBY;
      =     DBX [AR2,P#8.5];
      CDB;
      BLD   15;
NETWORK
TITLE = salida x12
      A     #X12;
      =     #EXPULSAR_PALET;
NETWORK
TITLE = salida x0
      A     #X0;
      =     #STBY;
NETWORK
TITLE =
      A     #RESET;
      R     #X11;
      R     #X12;
      S     #X0;
      R     #START_CIZA;
      R     #XERROR;
NETWORK
TITLE =
      A     #ERROR;
      R     #X11;
      R     #X12;
      R     #X0;
      R     #START_CIZA;
      S     #XERROR;
END_FUNCTION_BLOCK

FUNCTION_BLOCK "CORTA"	// FB 8
VERSION : 0.1
VAR_INPUT
  SENSORABAJO : BOOL ;
  SENSORARRIBA : BOOL ;
  EXPULSADA : BOOL ;
  START : BOOL ;
  OK : BOOL ;
  ERROR : BOOL ;
  RESET : BOOL ;
END_VAR
VAR_OUTPUT
  BAJARCUCHILLA : BOOL ;
  EXPULSARPLANCHA : BOOL ;
  BIT_OK : BOOL ;
  STBY : BOOL ;
END_VAR
VAR
  X51 : BOOL ;
  X52 : BOOL ;
  X53 : BOOL ;
  S3 : BOOL ;
  BDT : BOOL ;
  X50 : BOOL ;
  FP_START : BOOL ;
  XERROR : BOOL ;
END_VAR
BEGIN
NETWORK
TITLE = Arranque
      SET;
      FP    #BDT;
      S     #X50;
      R     #X51;
      R     #X52;
      R     #X53;
      R     #S3;
      R     #XERROR;
NETWORK
TITLE =
      A     #RESET;
      S     #X50;
      R     #X51;
      R     #X52;
      R     #X53;
      R     #S3;
      R     #XERROR;
NETWORK
TITLE =
      A     #ERROR;
      R     #X50;
      R     #X51;
      R     #X52;
      R     #X53;
      R     #S3;
      S     #XERROR;
NETWORK
TITLE = de x51 a x52
      A     #X51;
      A     #SENSORABAJO;
      R     #X51;
      S     #X52;
NETWORK
TITLE = de x52 a x53
      A     #X52;
      A     #SENSORARRIBA;
      R     #X52;
      S     #X53;
NETWORK
TITLE = de x53 a s3
      A     #X53;
      A     #EXPULSADA;
      R     #X53;
      S     #S3;
NETWORK
TITLE = Accion x51
      A     #X51;
      =     #BAJARCUCHILLA;
NETWORK
TITLE = Accion x53
      A     #X53;
      =     #EXPULSARPLANCHA;
NETWORK
TITLE = Accion final
      A     #S3;
      =     #BIT_OK;
NETWORK
TITLE = De s3 a x50
      A     #S3;
      A     #OK;
      R     #S3;
      S     #X50;
NETWORK
TITLE = De x50 a x51
      A     #X50;
      A     #START;
      FP    #FP_START;
      R     #X50;
      S     #X51;
NETWORK
TITLE = Salida x50
      A     #X50;
      =     #STBY;
END_FUNCTION_BLOCK

FUNCTION_BLOCK "MODO"	// FB 9
VERSION : 0.1
VAR_INPUT
  MODO1 : BOOL ;
  MODO2 : BOOL ;
END_VAR
VAR_OUTPUT
  STBY : BOOL ;
END_VAR
VAR
  X60 : BOOL ;
  X61 : BOOL ;
  X62 : BOOL ;
  BDT : BOOL ;
  FP_X61 : BOOL ;
  FP_X62 : BOOL ;
END_VAR
BEGIN
NETWORK
TITLE =
      SET;
      FP    #BDT;
      S     #X60;
      R     #X61;
      R     #X62;
NETWORK
TITLE =
      A     #X60;
      A     #MODO1;
      R     #X60;
      S     #X61;
NETWORK
TITLE =
      A     #X60;
      A     #MODO2;
      R     #X60;
      S     #X62;
NETWORK
TITLE =
      A     #X61;
      AN    #MODO1;
      R     #X61;
      S     #X60;
NETWORK
TITLE =
      A     #X62;
      AN    #MODO2;
      R     #X62;
      S     #X60;
NETWORK
TITLE =
      A     #X60;
      =     #STBY;
NETWORK
TITLE = Numero de planchas por bobina y peso Modo 1
      A     #X61;
      JCN   _001;
      L     "Modo1".PLANCHAS;
      T     "Global".PLANCHAS;
      L     "Modo1".PESO_PAELLERA;
      T     "Global".PESO_PAELLERA;
      L     "Modo1".PESO_WOK;
      T     "Global".PESO_WOK;
      L     "Modo1".PESO_SARTEN;
      T     "Global".PESO_SARTEN;
      L     "Modo1".PESO_CACEROLA;
      T     "Global".PESO_CACEROLA;
_001: NOP   0;
NETWORK
TITLE =
      A     #X62;
      JCN   _002;
      L     "Modo2".PLANCHAS;
      T     "Global".PLANCHAS;
      L     "Modo2".PESO_PAELLERA;
      T     "Global".PESO_PAELLERA;
      L     "Modo2".PESO_WOK;
      T     "Global".PESO_WOK;
      L     "Modo2".PESO_SARTEN;
      T     "Global".PESO_SARTEN;
      L     "Modo2".PESO_CACEROLA;
      T     "Global".PESO_CACEROLA;
_002: NOP   0;
END_FUNCTION_BLOCK

FUNCTION "ERRORES" : VOID	// FC 1
VERSION : 0.1
VAR_INPUT
  SENSORARRIBA : BOOL ;
  TEMP : TIMER ;
  RESET : BOOL ;
  SETA_PELIGROSA : BOOL ;
END_VAR
VAR_OUTPUT
  ERROR : BOOL ;
END_VAR
VAR_TEMP
  ERR1 : BOOL ;
  ERR2 : BOOL ;
  BDT : BOOL ;
END_VAR
BEGIN
NETWORK
TITLE =
      AN    #SENSORARRIBA;
      L     S5T#5S;
      SS    #TEMP;
NETWORK
TITLE =
      A     #SENSORARRIBA;
      R     #TEMP;
NETWORK
TITLE =
      A     #TEMP;
      =     #ERR1;
NETWORK
TITLE =
      A     #SETA_PELIGROSA;
      =     #ERR2;
NETWORK
TITLE =
      O     #ERR1;
      O     #ERR2;
      S     #ERROR;
NETWORK
TITLE =
      A     #RESET;
      R     #TEMP;
      R     #ERROR;
END_FUNCTION

FUNCTION "PESAJE" : VOID	// FC 2
TITLE = PESAJE
VERSION : 0.1
VAR_INPUT
  in : INT ;
  PESO_SARTEN : REAL ;
  PESO_CACEROLA : REAL ;
  PESO_WOK : REAL ;
  PESO_PAELLERA : REAL ;
  bit_de_trabajo : BOOL ;
  RECIBIDO : BOOL ;
  START : BOOL ;
END_VAR
VAR_OUTPUT
  stby : BOOL ;
  SARTEN : BOOL ;
  CACEROLA : BOOL ;
  WOK : BOOL ;
  PAELLERA : BOOL ;
  PESO_OUT : REAL ;
END_VAR
VAR_TEMP
  retFC105 : WORD ;
  x121 : BOOL ;
  x122 : BOOL ;
  x123 : BOOL ;
  x124 : BOOL ;
  m3 : BOOL ;
  x120 : BOOL ;
  FP_BDT : BOOL ;
  FP_START : BOOL ;
  PESO : REAL ;
END_VAR
BEGIN
NETWORK
TITLE = Pesado
      A     #m3;
      CALL  "SCALE" (
           $1                       := #in,
           $2                       := L#1133903872,
           $3                       := L#0,
           $4                       := FALSE,
           $5                       := #retFC105,
           $6                       := #PESO);
NETWORK
TITLE =
      A     #x120;
      A     #START;
      FP    #FP_START;
      R     #x120;
      S     #m3;
NETWORK
TITLE = Arranque
      A     #bit_de_trabajo;
      FP    #FP_BDT;
      S     #x120;
      R     #m3;
      R     #x121;
      R     #x122;
      R     #x123;
      R     #x124;
NETWORK
TITLE =
      A(;
      L     #PESO_SARTEN;
      L     5.000000e+00;
      +R;
      L     #PESO;
      >R;
      );
      A(;
      L     #PESO_SARTEN;
      L     5.000000e+00;
      -R;
      L     #PESO;
      <R;
      );
      A     #m3;
      R     #m3;
      S     #x121;
NETWORK
TITLE =
      L     #PESO;
      T     #PESO_OUT;
NETWORK
TITLE =
      A(;
      L     #PESO_CACEROLA;
      L     5.000000e+00;
      +R;
      L     #PESO;
      >R;
      );
      A(;
      L     #PESO_CACEROLA;
      L     5.000000e+00;
      -R;
      L     #PESO;
      <R;
      );
      A     #m3;
      R     #m3;
      S     #x122;
NETWORK
TITLE =
      A(;
      L     #PESO_WOK;
      L     5.000000e+00;
      +R;
      L     #PESO;
      >R;
      );
      A(;
      L     #PESO_WOK;
      L     5.000000e+00;
      -R;
      L     #PESO;
      <R;
      );
      A     #m3;
      R     #m3;
      S     #x123;
NETWORK
TITLE =
      A(;
      L     #PESO_PAELLERA;
      L     5.000000e+00;
      +R;
      L     #PESO;
      >R;
      );
      A(;
      L     #PESO_PAELLERA;
      L     5.000000e+00;
      -R;
      L     #PESO;
      <R;
      );
      A     #m3;
      R     #m3;
      S     #x124;
NETWORK
TITLE = TRATAMIENTO SALIDAS
      A     #x121;
      =     #SARTEN;
      A     #x122;
      =     #CACEROLA;
      A     #x123;
      =     #WOK;
      A     #x124;
      =     #PAELLERA;
      A     #x120;
      =     #stby;
NETWORK
TITLE = Paso de estado pesado a stby
      A(;
      A     #x121;
      O     #x122;
      O     #x123;
      O     #x124;
      );
      A     #RECIBIDO;
      R     #x121;
      R     #x122;
      R     #x123;
      R     #x124;
      S     #x120;
END_FUNCTION

// FC 105: know-how protected block, not included

DATA_BLOCK "Global"	// DB 1
VERSION : 0.1
  STRUCT
   PESO_CACEROLA : REAL  := 1.000000e+002;	//Peso Bobina Cacerolas
   PESO_WOK : REAL  := 1.100000e+002;	//Peso Bobina Wok
   PESO_SARTEN : REAL  := 1.200000e+002;	//Peso Bobina Sarten
   PESO_PAELLERA : REAL  := 1.300000e+002;	//Peso Bobina Paellera
   PLANCHAS : WORD  := W#16#100;	//Número de planchas por bobina
  END_STRUCT ;	
BEGIN
   PESO_CACEROLA := 1.000000e+02;
   PESO_WOK := 1.100000e+02;
   PESO_SARTEN := 1.200000e+02;
   PESO_PAELLERA := 1.300000e+02;
   PLANCHAS := W#16#100;
END_DATA_BLOCK

DATA_BLOCK "Modo1"	// DB 2
VERSION : 0.1
  STRUCT
   PESO_CACEROLA : REAL  := 1.100000e+002;	//Peso Bobina Cacerolas
   PESO_WOK : REAL  := 1.200000e+002;	//Peso Bobina Wok
   PESO_SARTEN : REAL  := 1.000000e+002;	//Peso Bobina Sarten
   PESO_PAELLERA : REAL  := 1.300000e+002;	//Peso Bobina Paellera
   PLANCHAS : WORD  := W#16#100;	//Número de planchas por bobina
  END_STRUCT ;	
BEGIN
   PESO_CACEROLA := 1.000000e+02;
   PESO_WOK := 1.100000e+02;
   PESO_SARTEN := 1.200000e+02;
   PESO_PAELLERA := 1.300000e+02;
   PLANCHAS := W#16#100;
END_DATA_BLOCK

DATA_BLOCK "Modo2"	// DB 3
VERSION : 0.1
  STRUCT
   PESO_CACEROLA : REAL  := 2.200000e+002;	//Peso Bobina Cacerolas
   PESO_WOK : REAL  := 2.400000e+002;	//Peso Bobina Wok
   PESO_SARTEN : REAL  := 2.000000e+002;	//Peso Bobina Sarten
   PESO_PAELLERA : REAL  := 2.600000e+002;	//Peso Bobina Paellera
   PLANCHAS : WORD  := W#16#200;	//Número de planchas por bobina
  END_STRUCT ;	
BEGIN
   PESO_CACEROLA := 2.000000e+02;
   PESO_WOK := 2.200000e+02;
   PESO_SARTEN := 2.400000e+02;
   PESO_PAELLERA := 2.600000e+02;
   PLANCHAS := W#16#200;
END_DATA_BLOCK

DATA_BLOCK "INFO_BOB"	// DB 4
VERSION : 0.1
  STRUCT
   CENTRO_CACEROLA : INT  := 20;
   CENTRO_SARTEN : INT  := 10;
   CENTRO_WOK : INT  := 30;
   CENTRO_PAELLERA : INT  := 40;
  END_STRUCT ;	
BEGIN
   CENTRO_CACEROLA := 20;
   CENTRO_SARTEN := 10;
   CENTRO_WOK := 30;
   CENTRO_PAELLERA := 40;
END_DATA_BLOCK

DATA_BLOCK DB 10
VERSION : 0.0
"GENERAL"
BEGIN
END_DATA_BLOCK

ORGANIZATION_BLOCK "CYCL_EXC"	// OB 1
TITLE = "Main Program Sweep (Cycle)"
VERSION : 0.1
VAR_TEMP
  OB1_EV_CLASS : BYTE ;	//Bits 0-3 = 1 (Coming event), Bits 4-7 = 1 (Event class 1)
  OB1_SCAN_1 : BYTE ;	//1 (Cold restart scan 1 of OB 1), 3 (Scan 2-n of OB 1)
  OB1_PRIORITY : BYTE ;	//Priority of OB Execution
  OB1_OB_NUMBR : BYTE ;	//1 (Organization block 1, OB1)
  OB1_RESERVED_1 : BYTE ;	//Reserved for system
  OB1_RESERVED_2 : BYTE ;	//Reserved for system
  OB1_PREV_CYCLE : INT ;	//Cycle time of previous OB1 scan (milliseconds)
  OB1_MIN_CYCLE : INT ;	//Minimum cycle time of OB1 (milliseconds)
  OB1_MAX_CYCLE : INT ;	//Maximum cycle time of OB1 (milliseconds)
  OB1_DATE_TIME : DATE_AND_TIME ;	//Date and time OB1 started
END_VAR
BEGIN
NETWORK
TITLE =
      CALL  "GENERAL" , DB 10 (
           BOBINA_COLOCADA          := "BOBINA_COLOCADA",
           MCENTRO                  := "MCENTRO",
           IN_PESAJE                := "IN_PESAJE",
           S_SARTEN                 := "S_SARTEN",
           S_CACEROLA               := "S_CACEROLA",
           S_WOK                    := "S_WOK",
           S_PAELLERA               := "S_PAELLERA",
           PRESENCIA                := "PRESENCIA",
           CONTADOR                 := "CONTADOR",
           PALET                    := "PALET",
           SENSORARRIBA             := "SENSORARRIBA",
           SENSORABAJO              := "SENSORABAJO",
           EXPULSADA                := "EXPULSADA",
           ON                       := "ON",
           MODO_1                   := "MODO_1",
           MODO_2                   := "MODO_2",
           ERROR                    := "ERROR",
           RESET                    := "RESET",
           PESO_OUT                 := "PESO_OUT",
           ABRIRMCENTRO             := "ABRIRMCENTRO",
           CERRARMCENTRO            := "CERRARMCENTRO",
           DESBOBINAR               := "DESBOBINAR",
           EXPULSAR_BOBINA          := "EXPULSAR_BOBINA",
           EXPULSAR_PLANCHA         := "EXPULSAR_PLANCHA",
           BAJAR_CUCHILLA           := "BAJAR_CUCHILLA",
           EXPULSAR_PALET           := "EXPULSAR_PALET",
           PRENSA                   := "PRENSA",
           STBY_DESBOB_1            := "STBY_DESBOB",
           STBY_CIZA_1              := "STBY_CIZA");
NETWORK
TITLE =
      CALL  "ERRORES" (
           SENSORARRIBA             := "SENSORARRIBA",
           TEMP                     := "TEMP_ERROR",
           RESET                    := "RESET",
           SETA_PELIGROSA           := "SETA_PELIGROSA",
           ERROR                    := "ERROR");
END_ORGANIZATION_BLOCK

SYMBOL_TABLE
"CONTADOR"	C 1	COUNTER
"DESBOBINADO"	FB 1	FB 1	// Función que se encarga del desbobinado
"SENSOR"	I 124.0	BOOL
"PRESENCIA"	I 124.1	BOOL
"START"	I 124.2	BOOL
"ERROR"	I 124.3	BOOL
"RESET"	I 124.4	BOOL
"BAJAR_CONT"	I 124.5	BOOL
"Cycle Execution"	OB 1	OB 1
"PLANCHAS"	PIW 651	WORD
"CENTRO"	PIW 653	INT
"MCENTRO"	PIW 655	INT
"ABRIRMCENTRO"	Q 100.0	BOOL
"DESBOBINAR"	Q 100.1	BOOL
"STBY"	Q 100.2	BOOL
END_SYMBOL_TABLE

FUNCTION_BLOCK "DESBOBINADO"	// FB 1
TITLE = DESBOBINADO
VERSION : 0.1
VAR_INPUT
  SENSOR : BOOL ;
  PRESENCIA : BOOL ;
  CENTRO : INT ;
  MCENTRO : INT ;
  Contador : COUNTER ;
  START : BOOL ;
  PLANCHAS : WORD  := W#16#100;
  ERROR : BOOL ;
  RESET : BOOL ;
END_VAR
VAR_OUTPUT
  ABRIRMCENTRO : BOOL ;
  DESBOBINAR : BOOL ;
  STBY : BOOL ;
END_VAR
VAR
  x31 : BOOL ;
  x32 : BOOL ;
  x33 : BOOL ;
  x34 : BOOL ;
  x30 : BOOL ;
  FP_PRESENCIA : BOOL ;
  BDT : BOOL ;
  FP_START : BOOL ;
  XERROR : BOOL ;
END_VAR
VAR_TEMP
  watchdog_master : BOOL ;
END_VAR
BEGIN
NETWORK
TITLE = Arranque
      SET;
      FP    #BDT;
      S     #x30;
      R     #x31;
      R     #x32;
      R     #x33;
      R     #x34;
NETWORK
TITLE =
      A     #RESET;
      R     #ABRIRMCENTRO;
      R     #DESBOBINAR;
      S     #x30;
      R     #x31;
      R     #x32;
      R     #x33;
      R     #x34;
      R     #XERROR;
NETWORK
TITLE =
      A     #ERROR;
      R     #ABRIRMCENTRO;
      R     #DESBOBINAR;
      R     #x30;
      R     #x31;
      R     #x32;
      R     #x33;
      R     #x34;
      S     #XERROR;
NETWORK
TITLE = x31 a x32
//Comparacion medida centro con medida nominal del centro para pasar de x31 a x32
      A     #x31;
      A(;
      L     #CENTRO;
      L     #MCENTRO;
      ==R;
      );
      R     #x31;
      S     #x32;
NETWORK
TITLE = x32 a x33
//Presencia detecta que la plancha esta en posicion para empezar el proceso de 
//desbobinado-cizallado
      A     #x32;
      A     #PRESENCIA;
      FP    #FP_PRESENCIA;
      R     #x32;
      S     #x33;
NETWORK
TITLE = x33 a x34
//Detecta que la plancha esta lista para ser cizallada
      A     #x33;
      A     #SENSOR;
      R     #x33;
      S     #x34;
NETWORK
TITLE = x34 a x33
//si el contador no ha acabado
      A     #x34;
      T     LD 1;
      TAK;
      T     LD 5;
      L     #Contador;
      T     LW 9;
      L     LD 5;
      L     LD 1;
      A     C [LW 9];
      AN    #SENSOR;
      R     #x34;
      S     #x33;
NETWORK
TITLE = x34 a X30
//si el contador ha cabado
      A     #x34;
      T     LD 1;
      TAK;
      T     LD 5;
      L     #Contador;
      T     LW 9;
      L     LD 5;
      L     LD 1;
      AN    C [LW 9];
      AN    #SENSOR;
      AN    #PRESENCIA;
      R     #x34;
      S     #x30;
NETWORK
TITLE = Tratamiento de bit de fin
      A     #x30;
      =     #STBY;
NETWORK
TITLE = Abrir centro
      A     #x31;
      =     #ABRIRMCENTRO;
NETWORK
TITLE = Carga del contador y desbobinado en x32
      A     #x32;
      S     #DESBOBINAR;
      L     #PLANCHAS;
      T     LD 1;
      TAK;
      T     LD 5;
      L     #Contador;
      T     LW 9;
      L     LD 5;
      L     LD 1;
      S     C [LW 9];
NETWORK
TITLE = Resta del contador y salida del x33
      A     #x33;
      S     #DESBOBINAR;
NETWORK
TITLE = Reset del desbobionado en x34
      A     #x34;
      R     #DESBOBINAR;
NETWORK
TITLE = De X30 a X31
      A     #START;
      FP    #FP_START;
      A     #x30;
      R     #x30;
      S     #x31;
END_FUNCTION_BLOCK

DATA_BLOCK DB 1
VERSION : 0.0
"DESBOBINADO"
BEGIN
END_DATA_BLOCK

ORGANIZATION_BLOCK "Cycle Execution"	// OB 1
TITLE = "Main Program Sweep (Cycle)"
VERSION : 0.1
VAR_TEMP
  OB1_EV_CLASS : BYTE ;	//Bits 0-3 = 1 (Coming event), Bits 4-7 = 1 (Event class 1)
  OB1_SCAN_1 : BYTE ;	//1 (Cold restart scan 1 of OB 1), 3 (Scan 2-n of OB 1)
  OB1_PRIORITY : BYTE ;	//Priority of OB Execution
  OB1_OB_NUMBR : BYTE ;	//1 (Organization block 1, OB1)
  OB1_RESERVED_1 : BYTE ;	//Reserved for system
  OB1_RESERVED_2 : BYTE ;	//Reserved for system
  OB1_PREV_CYCLE : INT ;	//Cycle time of previous OB1 scan (milliseconds)
  OB1_MIN_CYCLE : INT ;	//Minimum cycle time of OB1 (milliseconds)
  OB1_MAX_CYCLE : INT ;	//Maximum cycle time of OB1 (milliseconds)
  OB1_DATE_TIME : DATE_AND_TIME ;	//Date and time OB1 started
END_VAR
BEGIN
NETWORK
TITLE =
      A     "BAJAR_CONT";
      CD    "CONTADOR";
NETWORK
TITLE =
      CALL  "DESBOBINADO" , DB 1 (
           SENSOR                   := "SENSOR",
           PRESENCIA                := "PRESENCIA",
           CENTRO                   := "CENTRO",
           MCENTRO                  := "MCENTRO",
           Contador                 := "CONTADOR",
           START                    := "START",
           PLANCHAS                 := "PLANCHAS",
           ERROR                    := "ERROR",
           RESET                    := "RESET",
           ABRIRMCENTRO             := "ABRIRMCENTRO",
           DESBOBINAR               := "DESBOBINAR",
           STBY                     := "STBY");
END_ORGANIZATION_BLOCK

SYMBOL_TABLE
"CONTADOR"	C 1	COUNTER
"CIZALLADO"	FB 2	FB 2	// Funcion que se encaga del cizallado de planchas
"CORTA"	FB 8	FB 8
"CORTAR"	FC 1	FC 1	// Funcion de cortar las planchas
"RESET"	I 124.0	BOOL
"SENSOR"	I 124.1	BOOL
"SENSORABAJO"	I 124.2	BOOL
"SENSORARRIBA"	I 124.3	BOOL
"EXPULSADA"	I 124.4	BOOL
"START"	I 124.5	BOOL
"CARGAR_CONT"	I 124.6	BOOL
"ERROR"	I 124.7	BOOL
"Cycle Execution"	OB 1	OB 1
"PLANCHAS"	PIW 651	INT
"BAJARCUCHILLA"	Q 100.0	BOOL
"EXPULSARPLANCHA"	Q 100.1	BOOL
"BIT_OK"	Q 100.2	BOOL
"STBY"	Q 100.3	BOOL
END_SYMBOL_TABLE

FUNCTION_BLOCK "CIZALLADO"	// FB 2
TITLE = CIZALLADO
VERSION : 0.1
VAR_INPUT
  SENSOR : BOOL ;
  SENSORABAJO : BOOL ;
  SENSORARRIBA : BOOL ;
  EXPULSADA : BOOL ;
  CONTADOR : COUNTER ;
  START : BOOL ;
  RESET : BOOL ;
  ERROR : BOOL ;
END_VAR
VAR_OUTPUT
  BAJARCUCHILLA : BOOL ;
  EXPULSARPLANCHA : BOOL ;
  STBY : BOOL ;
  BIT_OK : BOOL ;
END_VAR
VAR
  X41 : BOOL ;
  M3 : BOOL ;
  X43 : BOOL ;
  BDT : BOOL ;
  FP_START : BOOL ;
  INICORTAR : BOOL ;
  S2 : BOOL ;
  OK_CORTAR : BOOL ;
  STBY_CORTAR : BOOL ;
  CORTADO : BOOL ;
  XERROR : BOOL ;
  CORTAR : FB 8;
END_VAR
BEGIN
NETWORK
TITLE = Arranque
      SET;
      FP    #BDT;
      S     #X41;
      R     #M3;
      R     #X43;
      R     #INICORTAR;
      R     #CORTADO;
      R     #BIT_OK;
      R     #S2;
NETWORK
TITLE = De x41 a M3
      A     #X41;
      A     #SENSOR;
      A     #STBY_CORTAR;
      A     #START;
      FP    #FP_START;
      R     #X41;
      S     #M3;
NETWORK
TITLE = De M3 a x43
      A     #M3;
      A     #CORTADO;
      R     #M3;
      S     #X43;
NETWORK
TITLE = de x43 a x41
      A     #X43;
      A     #STBY_CORTAR;
      T     LD 0;
      TAK;
      T     LD 4;
      L     #CONTADOR;
      T     LW 8;
      L     LD 4;
      L     LD 0;
      AN    C [LW 8];
      R     #X43;
      S     #S2;
NETWORK
TITLE = de x43 a X41
      A     #X43;
      A     #STBY_CORTAR;
      T     LD 0;
      TAK;
      T     LD 4;
      L     #CONTADOR;
      T     LW 8;
      L     LD 4;
      L     LD 0;
      A     C [LW 8];
      R     #X43;
      S     #X41;
NETWORK
TITLE = Call M3
      CALL  #CORTAR (
           SENSORABAJO              := #SENSORABAJO,
           SENSORARRIBA             := #SENSORARRIBA,
           EXPULSADA                := #EXPULSADA,
           START                    := #INICORTAR,
           OK                       := #OK_CORTAR,
           ERROR                    := #ERROR,
           RESET                    := #RESET,
           BAJARCUCHILLA            := #BAJARCUCHILLA,
           EXPULSARPLANCHA          := #EXPULSARPLANCHA,
           BIT_OK                   := #CORTADO,
           STBY                     := #STBY_CORTAR);
NETWORK
TITLE = De M3 a X43
      A     #M3;
      A     #CORTADO;
      R     #M3;
      S     #X43;
NETWORK
TITLE = Salida M3
      A     #M3;
      =     #INICORTAR;
NETWORK
TITLE = Cuenta el numero de planchas cortadas
      A     #X43;
      =     #OK_CORTAR;
      T     LD 0;
      TAK;
      T     LD 4;
      L     #CONTADOR;
      T     LW 8;
      L     LD 4;
      L     LD 0;
      CD    C [LW 8];
NETWORK
TITLE = Salida X41
      A     #X41;
      =     #STBY;
NETWORK
TITLE = Salida S2
      A     #S2;
      =     #BIT_OK;
NETWORK
TITLE =
      A     #RESET;
      S     #X41;
      R     #M3;
      R     #X43;
      R     #INICORTAR;
      R     #CORTADO;
      R     #BIT_OK;
      R     #S2;
      R     #XERROR;
NETWORK
TITLE =
      A     #ERROR;
      R     #X41;
      R     #M3;
      R     #X43;
      R     #INICORTAR;
      R     #CORTADO;
      R     #BIT_OK;
      R     #S2;
      S     #XERROR;
END_FUNCTION_BLOCK

FUNCTION_BLOCK "CORTA"	// FB 8
VERSION : 0.1
VAR_INPUT
  SENSORABAJO : BOOL ;
  SENSORARRIBA : BOOL ;
  EXPULSADA : BOOL ;
  START : BOOL ;
  OK : BOOL ;
  ERROR : BOOL ;
  RESET : BOOL ;
END_VAR
VAR_OUTPUT
  BAJARCUCHILLA : BOOL ;
  EXPULSARPLANCHA : BOOL ;
  BIT_OK : BOOL ;
  STBY : BOOL ;
END_VAR
VAR
  X51 : BOOL ;
  X52 : BOOL ;
  X53 : BOOL ;
  S3 : BOOL ;
  BDT : BOOL ;
  X50 : BOOL ;
  FP_START : BOOL ;
  XERROR : BOOL ;
END_VAR
BEGIN
NETWORK
TITLE = Arranque
      SET;
      FP    #BDT;
      S     #X50;
      R     #X51;
      R     #X52;
      R     #X53;
      R     #S3;
      R     #XERROR;
NETWORK
TITLE =
      A     #RESET;
      S     #X50;
      R     #X51;
      R     #X52;
      R     #X53;
      R     #S3;
      R     #XERROR;
NETWORK
TITLE =
      A     #ERROR;
      R     #X50;
      R     #X51;
      R     #X52;
      R     #X53;
      R     #S3;
      S     #XERROR;
NETWORK
TITLE = de x51 a x52
      A     #X51;
      A     #SENSORABAJO;
      R     #X51;
      S     #X52;
NETWORK
TITLE = de x52 a x53
      A     #X52;
      A     #SENSORARRIBA;
      R     #X52;
      S     #X53;
NETWORK
TITLE = de x53 a s3
      A     #X53;
      A     #EXPULSADA;
      R     #X53;
      S     #S3;
NETWORK
TITLE = Accion x51
      A     #X51;
      =     #BAJARCUCHILLA;
NETWORK
TITLE = Accion x53
      A     #X53;
      =     #EXPULSARPLANCHA;
NETWORK
TITLE = Accion final
      A     #S3;
      =     #BIT_OK;
NETWORK
TITLE = De s3 a x50
      A     #S3;
      A     #OK;
      R     #S3;
      S     #X50;
NETWORK
TITLE = De x50 a x51
      A     #X50;
      A     #START;
      FP    #FP_START;
      R     #X50;
      S     #X51;
NETWORK
TITLE = Salida x50
      A     #X50;
      =     #STBY;
END_FUNCTION_BLOCK

DATA_BLOCK DB 1
VERSION : 0.0
"CIZALLADO"
BEGIN
END_DATA_BLOCK

ORGANIZATION_BLOCK "Cycle Execution"	// OB 1
TITLE = "Main Program Sweep (Cycle)"
VERSION : 0.1
VAR_TEMP
  OB1_EV_CLASS : BYTE ;	//Bits 0-3 = 1 (Coming event), Bits 4-7 = 1 (Event class 1)
  OB1_SCAN_1 : BYTE ;	//1 (Cold restart scan 1 of OB 1), 3 (Scan 2-n of OB 1)
  OB1_PRIORITY : BYTE ;	//Priority of OB Execution
  OB1_OB_NUMBR : BYTE ;	//1 (Organization block 1, OB1)
  OB1_RESERVED_1 : BYTE ;	//Reserved for system
  OB1_RESERVED_2 : BYTE ;	//Reserved for system
  OB1_PREV_CYCLE : INT ;	//Cycle time of previous OB1 scan (milliseconds)
  OB1_MIN_CYCLE : INT ;	//Minimum cycle time of OB1 (milliseconds)
  OB1_MAX_CYCLE : INT ;	//Maximum cycle time of OB1 (milliseconds)
  OB1_DATE_TIME : DATE_AND_TIME ;	//Date and time OB1 started
END_VAR
BEGIN
NETWORK
TITLE =
      CALL  "CIZALLADO" , DB 1 (
           SENSOR                   := "SENSOR",
           SENSORABAJO              := "SENSORABAJO",
           SENSORARRIBA             := "SENSORARRIBA",
           EXPULSADA                := "EXPULSADA",
           CONTADOR                 := "CONTADOR",
           START                    := "START",
           RESET                    := "RESET",
           ERROR                    := "ERROR",
           BAJARCUCHILLA            := "BAJARCUCHILLA",
           EXPULSARPLANCHA          := "EXPULSARPLANCHA",
           STBY                     := "STBY",
           BIT_OK                   := "BIT_OK");
NETWORK
TITLE =
      A     "CARGAR_CONT";
      L     "PLANCHAS";
      S     "CONTADOR";
END_ORGANIZATION_BLOCK

SYMBOL_TABLE
"CONTADOR"	C 1	COUNTER
"DESBOBINADO"	FB 1	FB 1	// Función que se encarga del desbobinado
"MULT_DESBOB"	FB 3	FB 3
"S_CACEROLA"	I 124.0	BOOL
"S_SARTEN"	I 124.1	BOOL
"S_PAELLERA"	I 124.2	BOOL
"S_WOK"	I 124.3	BOOL
"PRESENCIA"	I 124.4	BOOL
"BIT_DE_TRABAJO"	I 124.5	BOOL
"START"	I 124.6	BOOL
"BAJAR_CONT"	I 124.7	BOOL
"SARTEN"	I 125.0	BOOL
"CACEROLA"	I 125.1	BOOL
"WOK"	I 125.2	BOOL
"PAELLERA"	I 125.3	BOOL
"ERROR"	I 125.4	BOOL
"RESET"	I 125.5	BOOL
"Cycle Execution"	OB 1	OB 1
"C_CACEROLA"	PIW 651	INT
"C_SARTEN"	PIW 653	INT
"C_WOK"	PIW 655	INT
"C_PAELLERA"	PIW 657	INT
"MCENTRO"	PIW 659	INT
"PLANCHAS"	PIW 661	WORD
"ABRIRMCENTRO"	Q 100.0	BOOL
"DESBOBINAR"	Q 100.1	BOOL
"BIT_OK"	Q 100.2	BOOL
"BIT_ERROR"	Q 100.3	BOOL
"STBY"	Q 100.4	BOOL
"STBY_SARTEN"	Q 101.0	BOOL
"STBY_CACEROLA"	Q 101.1	BOOL
"STBY_PAELLERA"	Q 101.2	BOOL
"STBY_WOK"	Q 101.3	BOOL
END_SYMBOL_TABLE

FUNCTION_BLOCK "DESBOBINADO"	// FB 1
TITLE = DESBOBINADO
VERSION : 0.1
VAR_INPUT
  SENSOR : BOOL ;
  PRESENCIA : BOOL ;
  CENTRO : INT ;
  MCENTRO : INT ;
  Contador : COUNTER ;
  START : BOOL ;
  PLANCHAS : WORD  := W#16#100;
  ERROR : BOOL ;
  RESET : BOOL ;
END_VAR
VAR_OUTPUT
  ABRIRMCENTRO : BOOL ;
  DESBOBINAR : BOOL ;
  STBY : BOOL ;
END_VAR
VAR
  x31 : BOOL ;
  x32 : BOOL ;
  x33 : BOOL ;
  x34 : BOOL ;
  x30 : BOOL ;
  FP_PRESENCIA : BOOL ;
  BDT : BOOL ;
  FP_START : BOOL ;
  XERROR : BOOL ;
END_VAR
VAR_TEMP
  watchdog_master : BOOL ;
END_VAR
BEGIN
NETWORK
TITLE = Arranque
      SET;
      FP    #BDT;
      S     #x30;
      R     #x31;
      R     #x32;
      R     #x33;
      R     #x34;
NETWORK
TITLE =
      A     #RESET;
      R     #ABRIRMCENTRO;
      R     #DESBOBINAR;
      S     #x30;
      R     #x31;
      R     #x32;
      R     #x33;
      R     #x34;
      R     #XERROR;
NETWORK
TITLE =
      A     #ERROR;
      R     #ABRIRMCENTRO;
      R     #DESBOBINAR;
      R     #x30;
      R     #x31;
      R     #x32;
      R     #x33;
      R     #x34;
      S     #XERROR;
NETWORK
TITLE = x31 a x32
//Comparacion medida centro con medida nominal del centro para pasar de x31 a x32
      A     #x31;
      A(;
      L     #CENTRO;
      L     #MCENTRO;
      ==R;
      );
      R     #x31;
      S     #x32;
NETWORK
TITLE = x32 a x33
//Presencia detecta que la plancha esta en posicion para empezar el proceso de 
//desbobinado-cizallado
      A     #x32;
      A     #PRESENCIA;
      FP    #FP_PRESENCIA;
      R     #x32;
      S     #x33;
NETWORK
TITLE = x33 a x34
//Detecta que la plancha esta lista para ser cizallada
      A     #x33;
      A     #SENSOR;
      R     #x33;
      S     #x34;
NETWORK
TITLE = x34 a x33
//si el contador no ha acabado
      A     #x34;
      T     LD 1;
      TAK;
      T     LD 5;
      L     #Contador;
      T     LW 9;
      L     LD 5;
      L     LD 1;
      A     C [LW 9];
      AN    #SENSOR;
      R     #x34;
      S     #x33;
NETWORK
TITLE = x34 a X30
//si el contador ha cabado
      A     #x34;
      T     LD 1;
      TAK;
      T     LD 5;
      L     #Contador;
      T     LW 9;
      L     LD 5;
      L     LD 1;
      AN    C [LW 9];
      AN    #SENSOR;
      AN    #PRESENCIA;
      R     #x34;
      S     #x30;
NETWORK
TITLE = Tratamiento de bit de fin
      A     #x30;
      =     #STBY;
NETWORK
TITLE = Abrir centro
      A     #x31;
      =     #ABRIRMCENTRO;
NETWORK
TITLE = Carga del contador y desbobinado en x32
      A     #x32;
      S     #DESBOBINAR;
      L     #PLANCHAS;
      T     LD 1;
      TAK;
      T     LD 5;
      L     #Contador;
      T     LW 9;
      L     LD 5;
      L     LD 1;
      S     C [LW 9];
NETWORK
TITLE = Resta del contador y salida del x33
      A     #x33;
      S     #DESBOBINAR;
NETWORK
TITLE = Reset del desbobionado en x34
      A     #x34;
      R     #DESBOBINAR;
NETWORK
TITLE = De X30 a X31
      A     #START;
      FP    #FP_START;
      A     #x30;
      R     #x30;
      S     #x31;
END_FUNCTION_BLOCK

FUNCTION_BLOCK "MULT_DESBOB"	// FB 3
VERSION : 0.1
VAR_INPUT
  S_CACEROLA : BOOL ;
  S_SARTEN : BOOL ;
  S_PAELLERA : BOOL ;
  S_WOK : BOOL ;
  PRESENCIA : BOOL ;
  C_CACEROLA : INT ;
  C_SARTEN : INT ;
  C_WOK : INT ;
  C_PAELLERA : INT ;
  MCENTRO : INT ;
  CONTADOR : COUNTER ;
  PLANCHAS : WORD ;
  SARTEN : BOOL ;
  CACEROLA : BOOL ;
  WOK : BOOL ;
  PAELLERA : BOOL ;
  START : BOOL ;
  ERROR : BOOL ;
  RESET : BOOL ;
END_VAR
VAR_OUTPUT
  ABRIRMCENTRO : BOOL ;
  DESBOBINAR : BOOL ;
  BIT_OK : BOOL ;
  BIT_ERROR : BOOL ;
  STBY : BOOL ;
  STBY_SAR : BOOL ;
  STBY_CAC : BOOL ;
  STBY_WOK : BOOL ;
  STBY_PAELL : BOOL ;
END_VAR
VAR
  START_SAR : BOOL ;
  START_CAC : BOOL ;
  START_WOK : BOOL ;
  START_PAELL : BOOL ;
  FP_BDT : BOOL ;
  X1 : BOOL ;
  X2 : BOOL ;
  X3 : BOOL ;
  X4 : BOOL ;
  X5 : BOOL ;
  X6 : BOOL ;
  BDT : BOOL ;
  FP_START : BOOL ;
  FLAG_DESB : BOOL ;
  FP_DESBOB : BOOL ;
  F_START : BOOL ;
  FN_BDT : BOOL ;
  FN_X1 : BOOL ;
  SAR_DESBOB : FB 1;
  CAC_DESBOB : FB 1;
  WOK_DESBOB : FB 1;
  PAELL_DESBOB : FB 1;
END_VAR
BEGIN
NETWORK
TITLE = call del x2
      A     #X2;
      JCN   _001;
      S     #BDT;
      BLD   14;
      =     L 6.0;
      L     DINO;
      T     LW 4;
      CDB;
      OPN   DI [LW 4];
      TAR2  LD 0;
      A     DBX [AR2,P#0.1];
      =     #SAR_DESBOB.SENSOR;
      A     DBX [AR2,P#0.4];
      =     #SAR_DESBOB.PRESENCIA;
      L     DBW [AR2,P#4.0];
      T     #SAR_DESBOB.CENTRO;
      L     DBW [AR2,P#10.0];
      T     #SAR_DESBOB.MCENTRO;
      L     DBW [AR2,P#12.0];
      T     #SAR_DESBOB.Contador;
      A     DBX [AR2,P#20.0];
      =     #SAR_DESBOB.START;
      L     DBW [AR2,P#14.0];
      T     #SAR_DESBOB.PLANCHAS;
      A     DBX [AR2,P#16.5];
      =     #SAR_DESBOB.ERROR;
      A     DBX [AR2,P#16.6];
      =     #SAR_DESBOB.RESET;
      +AR2  P#24.0;
      UC    "DESBOBINADO";
      LAR2  LD 0;
      A     #SAR_DESBOB.ABRIRMCENTRO;
      =     DBX [AR2,P#18.0];
      A     #SAR_DESBOB.DESBOBINAR;
      =     DBX [AR2,P#18.1];
      A     #SAR_DESBOB.STBY;
      =     DBX [AR2,P#18.5];
      CDB;
      BLD   15;
_001: NOP   0;
NETWORK
TITLE = call del x3
      A     #X3;
      JCN   _002;
      S     #BDT;
      BLD   14;
      =     L 6.0;
      L     DINO;
      T     LW 4;
      CDB;
      OPN   DI [LW 4];
      TAR2  LD 0;
      A     DBX [AR2,P#0.0];
      =     #CAC_DESBOB.SENSOR;
      A     DBX [AR2,P#0.4];
      =     #CAC_DESBOB.PRESENCIA;
      L     DBW [AR2,P#2.0];
      T     #CAC_DESBOB.CENTRO;
      L     DBW [AR2,P#10.0];
      T     #CAC_DESBOB.MCENTRO;
      L     DBW [AR2,P#12.0];
      T     #CAC_DESBOB.Contador;
      A     DBX [AR2,P#20.1];
      =     #CAC_DESBOB.START;
      L     DBW [AR2,P#14.0];
      T     #CAC_DESBOB.PLANCHAS;
      A     DBX [AR2,P#16.5];
      =     #CAC_DESBOB.ERROR;
      A     DBX [AR2,P#16.6];
      =     #CAC_DESBOB.RESET;
      +AR2  P#42.0;
      UC    "DESBOBINADO";
      LAR2  LD 0;
      A     #CAC_DESBOB.ABRIRMCENTRO;
      =     DBX [AR2,P#18.0];
      A     #CAC_DESBOB.DESBOBINAR;
      =     DBX [AR2,P#18.1];
      A     #CAC_DESBOB.STBY;
      =     DBX [AR2,P#18.6];
      CDB;
      BLD   15;
_002: NOP   0;
NETWORK
TITLE = call del x4
      A     #X4;
      JCN   _003;
      S     #BDT;
      BLD   14;
      =     L 6.0;
      L     DINO;
      T     LW 4;
      CDB;
      OPN   DI [LW 4];
      TAR2  LD 0;
      A     DBX [AR2,P#0.3];
      =     #WOK_DESBOB.SENSOR;
      A     DBX [AR2,P#0.4];
      =     #WOK_DESBOB.PRESENCIA;
      L     DBW [AR2,P#6.0];
      T     #WOK_DESBOB.CENTRO;
      L     DBW [AR2,P#10.0];
      T     #WOK_DESBOB.MCENTRO;
      L     DBW [AR2,P#12.0];
      T     #WOK_DESBOB.Contador;
      A     DBX [AR2,P#20.2];
      =     #WOK_DESBOB.START;
      L     DBW [AR2,P#14.0];
      T     #WOK_DESBOB.PLANCHAS;
      A     DBX [AR2,P#16.5];
      =     #WOK_DESBOB.ERROR;
      A     DBX [AR2,P#16.6];
      =     #WOK_DESBOB.RESET;
      +AR2  P#60.0;
      UC    "DESBOBINADO";
      LAR2  LD 0;
      A     #WOK_DESBOB.ABRIRMCENTRO;
      =     DBX [AR2,P#18.0];
      A     #WOK_DESBOB.DESBOBINAR;
      =     DBX [AR2,P#18.1];
      A     #WOK_DESBOB.STBY;
      =     DBX [AR2,P#18.7];
      CDB;
      BLD   15;
_003: NOP   0;
NETWORK
TITLE = call del x5
      A     #X5;
      JCN   _004;
      S     #BDT;
      BLD   14;
      =     L 6.0;
      L     DINO;
      T     LW 4;
      CDB;
      OPN   DI [LW 4];
      TAR2  LD 0;
      A     DBX [AR2,P#0.2];
      =     #PAELL_DESBOB.SENSOR;
      A     DBX [AR2,P#0.4];
      =     #PAELL_DESBOB.PRESENCIA;
      L     DBW [AR2,P#8.0];
      T     #PAELL_DESBOB.CENTRO;
      L     DBW [AR2,P#10.0];
      T     #PAELL_DESBOB.MCENTRO;
      L     DBW [AR2,P#12.0];
      T     #PAELL_DESBOB.Contador;
      A     DBX [AR2,P#20.3];
      =     #PAELL_DESBOB.START;
      L     DBW [AR2,P#14.0];
      T     #PAELL_DESBOB.PLANCHAS;
      A     DBX [AR2,P#16.5];
      =     #PAELL_DESBOB.ERROR;
      A     DBX [AR2,P#16.6];
      =     #PAELL_DESBOB.RESET;
      +AR2  P#78.0;
      UC    "DESBOBINADO";
      LAR2  LD 0;
      A     #PAELL_DESBOB.ABRIRMCENTRO;
      =     DBX [AR2,P#18.0];
      A     #PAELL_DESBOB.DESBOBINAR;
      =     DBX [AR2,P#18.1];
      A     #PAELL_DESBOB.STBY;
      =     DBX [AR2,P#18.4];
      CDB;
      BLD   15;
_004: NOP   0;
NETWORK
TITLE = salida x2
      A     #X2;
      =     #START_SAR;
NETWORK
TITLE = salida x3
      A     #X3;
      =     #START_CAC;
NETWORK
TITLE = salida x4
      A     #X4;
      =     #START_WOK;
NETWORK
TITLE = salida x5
      A     #X5;
      =     #START_PAELL;
NETWORK
TITLE = Arranque
      SET;
      FP    #FP_BDT;
      R     #START_SAR;
      R     #START_CAC;
      R     #START_WOK;
      R     #START_PAELL;
      S     #X1;
      R     #X2;
      R     #X3;
      R     #X4;
      R     #X5;
      R     #X6;
NETWORK
TITLE = guardado de flanco de start
      A     #START;
      FP    #FP_START;
      =     #F_START;
NETWORK
TITLE = de x1 x2
      A     #F_START;
      A     #X1;
      A     #SARTEN;
      R     #X1;
      S     #X2;
NETWORK
TITLE = de x1 a x3
      A     #F_START;
      A     #X1;
      A     #CACEROLA;
      R     #X1;
      S     #X3;
NETWORK
TITLE = de x1 a x4
      A     #F_START;
      A     #X1;
      A     #WOK;
      R     #X1;
      S     #X4;
NETWORK
TITLE = de x1 a x5
      A     #F_START;
      A     #X1;
      A     #PAELLERA;
      R     #X1;
      S     #X5;
NETWORK
TITLE = Guardado flag desbobinado
      A     #DESBOBINAR;
      FP    #FP_DESBOB;
      S     #FLAG_DESB;
NETWORK
TITLE = de x2 a x6
      A     #X2;
      A     #FLAG_DESB;
      A     #STBY_SAR;
      R     #FLAG_DESB;
      R     #X2;
      S     #X6;
NETWORK
TITLE = de x3 a x6
      A     #X3;
      A     #FLAG_DESB;
      A     #STBY_CAC;
      R     #FLAG_DESB;
      R     #X3;
      S     #X6;
NETWORK
TITLE = de x4 a x6
      A     #X4;
      A     #FLAG_DESB;
      A     #STBY_WOK;
      R     #FLAG_DESB;
      R     #X4;
      S     #X6;
NETWORK
TITLE = de x5 a x6
      A     #X5;
      A     #FLAG_DESB;
      A     #STBY_PAELL;
      R     #FLAG_DESB;
      R     #X5;
      S     #X6;
NETWORK
TITLE = salida x1
      A     #X1;
      =     #STBY;
NETWORK
TITLE = salida x6 
      A     #X6;
      =     #BIT_OK;
NETWORK
TITLE = error, sin prgramar
      A     #RESET;
      A(;
      A(;
      O(;
      A     #STBY_CAC;
      A     #X3;
      );
      O(;
      A     #STBY_SAR;
      A     #X2;
      );
      O(;
      A     #STBY_WOK;
      A     #X4;
      );
      O(;
      A     #STBY_PAELL;
      A     #X5;
      );
      );
      O     #X6;
      );
      R     #BDT;
      R     #BIT_OK;
      R     #BIT_ERROR;
      S     #X1;
      R     #X2;
      R     #X3;
      R     #X4;
      R     #X5;
      R     #X6;
      R     #START_SAR;
      R     #START_CAC;
      R     #START_WOK;
      R     #START_PAELL;
      R     #FLAG_DESB;
      R     #ABRIRMCENTRO;
      R     #DESBOBINAR;
END_FUNCTION_BLOCK

DATA_BLOCK DB 1
VERSION : 0.0
"MULT_DESBOB"
BEGIN
END_DATA_BLOCK

ORGANIZATION_BLOCK "Cycle Execution"	// OB 1
TITLE = "Main Program Sweep (Cycle)"
VERSION : 0.1
VAR_TEMP
  OB1_EV_CLASS : BYTE ;	//Bits 0-3 = 1 (Coming event), Bits 4-7 = 1 (Event class 1)
  OB1_SCAN_1 : BYTE ;	//1 (Cold restart scan 1 of OB 1), 3 (Scan 2-n of OB 1)
  OB1_PRIORITY : BYTE ;	//Priority of OB Execution
  OB1_OB_NUMBR : BYTE ;	//1 (Organization block 1, OB1)
  OB1_RESERVED_1 : BYTE ;	//Reserved for system
  OB1_RESERVED_2 : BYTE ;	//Reserved for system
  OB1_PREV_CYCLE : INT ;	//Cycle time of previous OB1 scan (milliseconds)
  OB1_MIN_CYCLE : INT ;	//Minimum cycle time of OB1 (milliseconds)
  OB1_MAX_CYCLE : INT ;	//Maximum cycle time of OB1 (milliseconds)
  OB1_DATE_TIME : DATE_AND_TIME ;	//Date and time OB1 started
END_VAR
BEGIN
NETWORK
TITLE =
      SET;
      CALL  "MULT_DESBOB" , DB 1 (
           S_CACEROLA               := "S_CACEROLA",
           S_SARTEN                 := "S_SARTEN",
           S_PAELLERA               := "S_PAELLERA",
           S_WOK                    := "S_WOK",
           PRESENCIA                := "PRESENCIA",
           C_CACEROLA               := "C_CACEROLA",
           C_SARTEN                 := "C_SARTEN",
           C_WOK                    := "C_WOK",
           C_PAELLERA               := "C_PAELLERA",
           MCENTRO                  := "MCENTRO",
           CONTADOR                 := "CONTADOR",
           PLANCHAS                 := "PLANCHAS",
           SARTEN                   := "SARTEN",
           CACEROLA                 := "CACEROLA",
           WOK                      := "WOK",
           PAELLERA                 := "PAELLERA",
           START                    := "START",
           ERROR                    := "ERROR",
           RESET                    := "RESET",
           ABRIRMCENTRO             := "ABRIRMCENTRO",
           DESBOBINAR               := "DESBOBINAR",
           BIT_OK                   := "BIT_OK",
           BIT_ERROR                := "BIT_ERROR",
           STBY                     := "STBY",
           STBY_SAR                 := "STBY_SARTEN",
           STBY_CAC                 := "STBY_CACEROLA",
           STBY_WOK                 := "STBY_WOK",
           STBY_PAELL               := "STBY_PAELLERA");
NETWORK
TITLE =
      A     "BAJAR_CONT";
      CD    "CONTADOR";
END_ORGANIZATION_BLOCK

SYMBOL_TABLE
"CONTADOR"	C 1	COUNTER
"CIZALLADO"	FB 2	FB 2	// Funcion que se encaga del cizallado de planchas
"MULT_CIZA"	FB 4	FB 4
"CORTA"	FB 8	FB 8
"CORTAR"	FC 1	FC 1	// Funcion de cortar las planchas
"S_CACEROLA"	I 124.0	BOOL
"S_SARTEN"	I 124.1	BOOL
"S_PAELLERA"	I 124.2	BOOL
"S_WOK"	I 124.3	BOOL
"ERROR"	I 124.4	BOOL
"SENSORARRIBA"	I 124.6	BOOL
"SENSORABAJO"	I 124.7	BOOL
"EXPULSADA"	I 125.0	BOOL
"START"	I 125.1	BOOL
"LOAD_CONT"	I 125.2	BOOL
"SARTEN"	I 125.3	BOOL
"CACEROLA"	I 125.4	BOOL
"WOK"	I 125.5	BOOL
"PAELLERA"	I 125.6	BOOL
"RESET"	I 125.7	BOOL
"Cycle Execution"	OB 1	OB 1
"PLANCHAS"	PIW 651	INT
"EXPULSARPLANCHA"	Q 100.1	BOOL
"BAJARCUCHILLA"	Q 100.2	BOOL
"BIT_OK"	Q 100.3	BOOL
"STBY"	Q 100.4	BOOL
END_SYMBOL_TABLE

FUNCTION_BLOCK "CIZALLADO"	// FB 2
TITLE = CIZALLADO
VERSION : 0.1
VAR_INPUT
  SENSOR : BOOL ;
  SENSORABAJO : BOOL ;
  SENSORARRIBA : BOOL ;
  EXPULSADA : BOOL ;
  CONTADOR : COUNTER ;
  START : BOOL ;
  RESET : BOOL ;
  ERROR : BOOL ;
END_VAR
VAR_OUTPUT
  BAJARCUCHILLA : BOOL ;
  EXPULSARPLANCHA : BOOL ;
  STBY : BOOL ;
  BIT_OK : BOOL ;
END_VAR
VAR
  X41 : BOOL ;
  M3 : BOOL ;
  X43 : BOOL ;
  BDT : BOOL ;
  FP_START : BOOL ;
  INICORTAR : BOOL ;
  S2 : BOOL ;
  OK_CORTAR : BOOL ;
  STBY_CORTAR : BOOL ;
  CORTADO : BOOL ;
  XERROR : BOOL ;
  CORTAR : FB 8;
END_VAR
BEGIN
NETWORK
TITLE = Arranque
      SET;
      FP    #BDT;
      S     #X41;
      R     #M3;
      R     #X43;
      R     #INICORTAR;
      R     #CORTADO;
      R     #BIT_OK;
      R     #S2;
NETWORK
TITLE = De x41 a M3
      A     #X41;
      A     #SENSOR;
      A     #STBY_CORTAR;
      A     #START;
      FP    #FP_START;
      R     #X41;
      S     #M3;
NETWORK
TITLE = De M3 a x43
      A     #M3;
      A     #CORTADO;
      R     #M3;
      S     #X43;
NETWORK
TITLE = de x43 a x41
      A     #X43;
      A     #STBY_CORTAR;
      T     LD 0;
      TAK;
      T     LD 4;
      L     #CONTADOR;
      T     LW 8;
      L     LD 4;
      L     LD 0;
      AN    C [LW 8];
      R     #X43;
      S     #S2;
NETWORK
TITLE = de x43 a X41
      A     #X43;
      A     #STBY_CORTAR;
      T     LD 0;
      TAK;
      T     LD 4;
      L     #CONTADOR;
      T     LW 8;
      L     LD 4;
      L     LD 0;
      A     C [LW 8];
      R     #X43;
      S     #X41;
NETWORK
TITLE = Call M3
      CALL  #CORTAR (
           SENSORABAJO              := #SENSORABAJO,
           SENSORARRIBA             := #SENSORARRIBA,
           EXPULSADA                := #EXPULSADA,
           START                    := #INICORTAR,
           OK                       := #OK_CORTAR,
           ERROR                    := #ERROR,
           RESET                    := #RESET,
           BAJARCUCHILLA            := #BAJARCUCHILLA,
           EXPULSARPLANCHA          := #EXPULSARPLANCHA,
           BIT_OK                   := #CORTADO,
           STBY                     := #STBY_CORTAR);
NETWORK
TITLE = De M3 a X43
      A     #M3;
      A     #CORTADO;
      R     #M3;
      S     #X43;
NETWORK
TITLE = Salida M3
      A     #M3;
      =     #INICORTAR;
NETWORK
TITLE = Cuenta el numero de planchas cortadas
      A     #X43;
      =     #OK_CORTAR;
      T     LD 0;
      TAK;
      T     LD 4;
      L     #CONTADOR;
      T     LW 8;
      L     LD 4;
      L     LD 0;
      CD    C [LW 8];
NETWORK
TITLE = Salida X41
      A     #X41;
      =     #STBY;
NETWORK
TITLE = Salida S2
      A     #S2;
      =     #BIT_OK;
NETWORK
TITLE =
      A     #RESET;
      S     #X41;
      R     #M3;
      R     #X43;
      R     #INICORTAR;
      R     #CORTADO;
      R     #BIT_OK;
      R     #S2;
      R     #XERROR;
NETWORK
TITLE =
      A     #ERROR;
      R     #X41;
      R     #M3;
      R     #X43;
      R     #INICORTAR;
      R     #CORTADO;
      R     #BIT_OK;
      R     #S2;
      S     #XERROR;
END_FUNCTION_BLOCK

FUNCTION_BLOCK "MULT_CIZA"	// FB 4
VERSION : 0.1
VAR_INPUT
  S_CACEROLA : BOOL ;
  S_WOK : BOOL ;
  S_SARTEN : BOOL ;
  S_PAELLERA : BOOL ;
  SENSORARRIBA : BOOL ;
  SENSORABAJO : BOOL ;
  EXPULSADA : BOOL ;
  CONTADOR : COUNTER ;
  SARTEN : BOOL ;
  CACEROLA : BOOL ;
  WOK : BOOL ;
  PAELLERA : BOOL ;
  START : BOOL ;
  ERROR : BOOL ;
  RESET : BOOL ;
END_VAR
VAR_OUTPUT
  EXPULSARPLANCHA : BOOL ;
  BAJARCUCHILLA : BOOL ;
  BIT_OK : BOOL ;
  STBY : BOOL ;
END_VAR
VAR
  START_SAR : BOOL ;
  START_CAC : BOOL ;
  START_WOK : BOOL ;
  START_PAELL : BOOL ;
  X1 : BOOL ;
  X2 : BOOL ;
  X3 : BOOL ;
  X4 : BOOL ;
  X5 : BOOL ;
  FP_START : BOOL ;
  F_START : BOOL ;
  STBY_SAR : BOOL ;
  STBY_CAC : BOOL ;
  STBY_WOK : BOOL ;
  STBY_PAELL : BOOL ;
  OK : BOOL ;
  BDT : BOOL ;
  X6 : BOOL ;
  RESET_CIZA : BOOL ;
  FP_RESET : BOOL ;
  CAC_CIZA : FB 2;
  SAR_CIZA : FB 2;
  WOK_CIZA : FB 2;
  PAELL_CIZA : FB 2;
END_VAR
BEGIN
NETWORK
TITLE = Arranque
      SET;
      FP    #BDT;
      S     #X1;
      R     #X2;
      R     #X3;
      R     #X4;
      R     #X5;
      R     #X6;
NETWORK
TITLE = De x1 a x2
      A     #START;
      A     #SARTEN;
      A     #X1;
      R     #X1;
      S     #X2;
NETWORK
TITLE = de x1 a x3
      A     #START;
      A     #CACEROLA;
      A     #X1;
      R     #X1;
      S     #X3;
NETWORK
TITLE = de x1 a x4
      A     #START;
      A     #WOK;
      A     #X1;
      R     #X1;
      S     #X4;
NETWORK
TITLE = de x1 a x5
      A     #START;
      A     #PAELLERA;
      A     #X1;
      R     #X1;
      S     #X5;
NETWORK
TITLE = de x2-5 a x1
      A     #OK;
      A(;
      O     #X2;
      O     #X3;
      O     #X4;
      O     #X5;
      );
      R     #X2;
      R     #X3;
      R     #X4;
      R     #X5;
      S     #X1;
NETWORK
TITLE = call del x2
      A     #X2;
      JCN   _001;
      BLD   14;
      =     L 6.0;
      L     DINO;
      T     LW 4;
      CDB;
      OPN   DI [LW 4];
      TAR2  LD 0;
      A     DBX [AR2,P#0.2];
      =     #SAR_CIZA.SENSOR;
      A     DBX [AR2,P#0.5];
      =     #SAR_CIZA.SENSORABAJO;
      A     DBX [AR2,P#0.4];
      =     #SAR_CIZA.SENSORARRIBA;
      A     DBX [AR2,P#0.6];
      =     #SAR_CIZA.EXPULSADA;
      L     DBW [AR2,P#2.0];
      T     #SAR_CIZA.CONTADOR;
      A     DBX [AR2,P#8.0];
      =     #SAR_CIZA.START;
      A     DBX [AR2,P#10.2];
      =     #SAR_CIZA.RESET;
      A     DBX [AR2,P#4.5];
      =     #SAR_CIZA.ERROR;
      +AR2  P#28.0;
      UC    "CIZALLADO";
      LAR2  LD 0;
      A     #SAR_CIZA.BAJARCUCHILLA;
      =     DBX [AR2,P#6.1];
      A     #SAR_CIZA.EXPULSARPLANCHA;
      =     DBX [AR2,P#6.0];
      A     #SAR_CIZA.STBY;
      =     DBX [AR2,P#9.3];
      A     #SAR_CIZA.BIT_OK;
      =     DBX [AR2,P#9.7];
      CDB;
      BLD   15;
_001: NOP   0;
NETWORK
TITLE = call del x3
      A     #X3;
      JCN   _002;
      BLD   14;
      =     L 6.0;
      L     DINO;
      T     LW 4;
      CDB;
      OPN   DI [LW 4];
      TAR2  LD 0;
      A     DBX [AR2,P#0.0];
      =     #CAC_CIZA.SENSOR;
      A     DBX [AR2,P#0.5];
      =     #CAC_CIZA.SENSORABAJO;
      A     DBX [AR2,P#0.4];
      =     #CAC_CIZA.SENSORARRIBA;
      A     DBX [AR2,P#0.6];
      =     #CAC_CIZA.EXPULSADA;
      L     DBW [AR2,P#2.0];
      T     #CAC_CIZA.CONTADOR;
      A     DBX [AR2,P#8.1];
      =     #CAC_CIZA.START;
      A     DBX [AR2,P#10.2];
      =     #CAC_CIZA.RESET;
      A     DBX [AR2,P#4.5];
      =     #CAC_CIZA.ERROR;
      +AR2  P#12.0;
      UC    "CIZALLADO";
      LAR2  LD 0;
      A     #CAC_CIZA.BAJARCUCHILLA;
      =     DBX [AR2,P#6.1];
      A     #CAC_CIZA.EXPULSARPLANCHA;
      =     DBX [AR2,P#6.0];
      A     #CAC_CIZA.STBY;
      =     DBX [AR2,P#9.4];
      A     #CAC_CIZA.BIT_OK;
      =     DBX [AR2,P#9.7];
      CDB;
      BLD   15;
_002: NOP   0;
NETWORK
TITLE = call del x4
      A     #X4;
      JCN   _003;
      BLD   14;
      =     L 6.0;
      L     DINO;
      T     LW 4;
      CDB;
      OPN   DI [LW 4];
      TAR2  LD 0;
      A     DBX [AR2,P#0.1];
      =     #WOK_CIZA.SENSOR;
      A     DBX [AR2,P#0.5];
      =     #WOK_CIZA.SENSORABAJO;
      A     DBX [AR2,P#0.4];
      =     #WOK_CIZA.SENSORARRIBA;
      A     DBX [AR2,P#0.6];
      =     #WOK_CIZA.EXPULSADA;
      L     DBW [AR2,P#2.0];
      T     #WOK_CIZA.CONTADOR;
      A     DBX [AR2,P#8.2];
      =     #WOK_CIZA.START;
      A     DBX [AR2,P#10.2];
      =     #WOK_CIZA.RESET;
      A     DBX [AR2,P#4.5];
      =     #WOK_CIZA.ERROR;
      +AR2  P#44.0;
      UC    "CIZALLADO";
      LAR2  LD 0;
      A     #WOK_CIZA.BAJARCUCHILLA;
      =     DBX [AR2,P#6.1];
      A     #WOK_CIZA.EXPULSARPLANCHA;
      =     DBX [AR2,P#6.0];
      A     #WOK_CIZA.STBY;
      =     DBX [AR2,P#9.5];
      A     #WOK_CIZA.BIT_OK;
      =     DBX [AR2,P#9.7];
      CDB;
      BLD   15;
_003: NOP   0;
NETWORK
TITLE = call del x5
      A     #X5;
      JCN   _004;
      BLD   14;
      =     L 6.0;
      L     DINO;
      T     LW 4;
      CDB;
      OPN   DI [LW 4];
      TAR2  LD 0;
      A     DBX [AR2,P#0.3];
      =     #PAELL_CIZA.SENSOR;
      A     DBX [AR2,P#0.5];
      =     #PAELL_CIZA.SENSORABAJO;
      A     DBX [AR2,P#0.4];
      =     #PAELL_CIZA.SENSORARRIBA;
      A     DBX [AR2,P#0.6];
      =     #PAELL_CIZA.EXPULSADA;
      L     DBW [AR2,P#2.0];
      T     #PAELL_CIZA.CONTADOR;
      A     DBX [AR2,P#8.3];
      =     #PAELL_CIZA.START;
      A     DBX [AR2,P#10.2];
      =     #PAELL_CIZA.RESET;
      A     DBX [AR2,P#4.5];
      =     #PAELL_CIZA.ERROR;
      +AR2  P#60.0;
      UC    "CIZALLADO";
      LAR2  LD 0;
      A     #PAELL_CIZA.BAJARCUCHILLA;
      =     DBX [AR2,P#6.1];
      A     #PAELL_CIZA.EXPULSARPLANCHA;
      =     DBX [AR2,P#6.0];
      A     #PAELL_CIZA.STBY;
      =     DBX [AR2,P#9.6];
      A     #PAELL_CIZA.BIT_OK;
      =     DBX [AR2,P#9.7];
      CDB;
      BLD   15;
_004: NOP   0;
NETWORK
TITLE = salida x2
      A     #X2;
      =     #START_SAR;
NETWORK
TITLE = salida x3
      A     #X3;
      =     #START_CAC;
NETWORK
TITLE = salida x4
      A     #X4;
      =     #START_WOK;
NETWORK
TITLE = salida x5
      A     #X5;
      =     #START_PAELL;
NETWORK
TITLE =
      A     #X1;
      =     #STBY;
NETWORK
TITLE =
      A(;
      O     #X2;
      O     #X3;
      O     #X4;
      O     #X5;
      );
      FP    #FP_RESET;
      =     #RESET_CIZA;
NETWORK
TITLE =
      A     #RESET;
      A(;
      A(;
      O(;
      A     #STBY_CAC;
      A     #X3;
      );
      O(;
      A     #STBY_SAR;
      A     #X2;
      );
      O(;
      A     #STBY_WOK;
      A     #X4;
      );
      O(;
      A     #STBY_PAELL;
      A     #X5;
      );
      );
      O     #X6;
      );
      S     #X1;
      R     #X2;
      R     #X3;
      R     #X4;
      R     #X5;
      R     #EXPULSARPLANCHA;
      R     #BAJARCUCHILLA;
      R     #BIT_OK;
END_FUNCTION_BLOCK

FUNCTION_BLOCK "CORTA"	// FB 8
VERSION : 0.1
VAR_INPUT
  SENSORABAJO : BOOL ;
  SENSORARRIBA : BOOL ;
  EXPULSADA : BOOL ;
  START : BOOL ;
  OK : BOOL ;
  ERROR : BOOL ;
  RESET : BOOL ;
END_VAR
VAR_OUTPUT
  BAJARCUCHILLA : BOOL ;
  EXPULSARPLANCHA : BOOL ;
  BIT_OK : BOOL ;
  STBY : BOOL ;
END_VAR
VAR
  X51 : BOOL ;
  X52 : BOOL ;
  X53 : BOOL ;
  S3 : BOOL ;
  BDT : BOOL ;
  X50 : BOOL ;
  FP_START : BOOL ;
  XERROR : BOOL ;
END_VAR
BEGIN
NETWORK
TITLE = Arranque
      SET;
      FP    #BDT;
      S     #X50;
      R     #X51;
      R     #X52;
      R     #X53;
      R     #S3;
      R     #XERROR;
NETWORK
TITLE =
      A     #RESET;
      S     #X50;
      R     #X51;
      R     #X52;
      R     #X53;
      R     #S3;
      R     #XERROR;
NETWORK
TITLE =
      A     #ERROR;
      R     #X50;
      R     #X51;
      R     #X52;
      R     #X53;
      R     #S3;
      S     #XERROR;
NETWORK
TITLE = de x51 a x52
      A     #X51;
      A     #SENSORABAJO;
      R     #X51;
      S     #X52;
NETWORK
TITLE = de x52 a x53
      A     #X52;
      A     #SENSORARRIBA;
      R     #X52;
      S     #X53;
NETWORK
TITLE = de x53 a s3
      A     #X53;
      A     #EXPULSADA;
      R     #X53;
      S     #S3;
NETWORK
TITLE = Accion x51
      A     #X51;
      =     #BAJARCUCHILLA;
NETWORK
TITLE = Accion x53
      A     #X53;
      =     #EXPULSARPLANCHA;
NETWORK
TITLE = Accion final
      A     #S3;
      =     #BIT_OK;
NETWORK
TITLE = De s3 a x50
      A     #S3;
      A     #OK;
      R     #S3;
      S     #X50;
NETWORK
TITLE = De x50 a x51
      A     #X50;
      A     #START;
      FP    #FP_START;
      R     #X50;
      S     #X51;
NETWORK
TITLE = Salida x50
      A     #X50;
      =     #STBY;
END_FUNCTION_BLOCK

DATA_BLOCK DB 1
VERSION : 0.0
"MULT_CIZA"
BEGIN
END_DATA_BLOCK

ORGANIZATION_BLOCK "Cycle Execution"	// OB 1
TITLE = "Main Program Sweep (Cycle)"
VERSION : 0.1
VAR_TEMP
  OB1_EV_CLASS : BYTE ;	//Bits 0-3 = 1 (Coming event), Bits 4-7 = 1 (Event class 1)
  OB1_SCAN_1 : BYTE ;	//1 (Cold restart scan 1 of OB 1), 3 (Scan 2-n of OB 1)
  OB1_PRIORITY : BYTE ;	//Priority of OB Execution
  OB1_OB_NUMBR : BYTE ;	//1 (Organization block 1, OB1)
  OB1_RESERVED_1 : BYTE ;	//Reserved for system
  OB1_RESERVED_2 : BYTE ;	//Reserved for system
  OB1_PREV_CYCLE : INT ;	//Cycle time of previous OB1 scan (milliseconds)
  OB1_MIN_CYCLE : INT ;	//Minimum cycle time of OB1 (milliseconds)
  OB1_MAX_CYCLE : INT ;	//Maximum cycle time of OB1 (milliseconds)
  OB1_DATE_TIME : DATE_AND_TIME ;	//Date and time OB1 started
END_VAR
BEGIN
NETWORK
TITLE =
      CALL  "MULT_CIZA" , DB 1 (
           S_CACEROLA               := "S_CACEROLA",
           S_WOK                    := "S_WOK",
           S_SARTEN                 := "S_SARTEN",
           S_PAELLERA               := "S_PAELLERA",
           SENSORARRIBA             := "SENSORARRIBA",
           SENSORABAJO              := "SENSORABAJO",
           EXPULSADA                := "EXPULSADA",
           CONTADOR                 := "CONTADOR",
           SARTEN                   := "SARTEN",
           CACEROLA                 := "CACEROLA",
           WOK                      := "WOK",
           PAELLERA                 := "PAELLERA",
           START                    := "START",
           ERROR                    := "ERROR",
           RESET                    := "RESET",
           EXPULSARPLANCHA          := "EXPULSARPLANCHA",
           BAJARCUCHILLA            := "BAJARCUCHILLA",
           BIT_OK                   := "BIT_OK",
           STBY                     := "STBY");
NETWORK
TITLE =
      A     "LOAD_CONT";
      JCN   _010;
      L     "PLANCHAS";
      S     "CONTADOR";
_010: NOP   0;
END_ORGANIZATION_BLOCK

SYMBOL_TABLE
"CONTADOR"	C 1	COUNTER
"Global"	DB 1	DB 1
"INFO_BOB"	DB 4	DB 4
"DESBOBINADO"	FB 1	FB 1	// Función que se encarga del desbobinado
"MULT_DESBOB"	FB 3	FB 3
"MULT_GEN_DESB"	FB 6	FB 6
"PESAJE"	FC 2	FC 2	// Función de pesaje
"SCALE"	FC 105	FC 105	// Scaling Values
"START"	I 124.0	BOOL
"ERROR"	I 124.1	BOOL
"BOBINA_COLOCADA"	I 124.2	BOOL
"S_SARTEN"	I 124.3	BOOL
"S_CACEROLA"	I 124.4	BOOL
"S_WOK"	I 124.5	BOOL
"S_PAELLERA"	I 124.6	BOOL
"PRESENCIA"	I 124.7	BOOL
"RESET"	I 125.0	BOOL
"SARTEN"	M 120.0	BOOL
"CACEROLA"	M 120.1	BOOL
"WOK"	M 120.2	BOOL
"PAELLERA"	M 120.3	BOOL
"PESO_OUT"	MD 100	REAL
"Cycle Execution"	OB 1	OB 1
"MCENTRO"	PIW 751	INT
"IN_PESAJE"	PIW 753	INT
"ABRIRMCENTRO"	Q 100.0	BOOL
"CERRARMCENTRO"	Q 100.1	BOOL
"DESBOBINAR"	Q 100.2	BOOL
"EXPULSAR_BOBINA"	Q 100.3	BOOL
"STBY"	Q 100.4	BOOL
END_SYMBOL_TABLE

FUNCTION_BLOCK "DESBOBINADO"	// FB 1
TITLE = DESBOBINADO
VERSION : 0.1
VAR_INPUT
  SENSOR : BOOL ;
  PRESENCIA : BOOL ;
  CENTRO : INT ;
  MCENTRO : INT ;
  Contador : COUNTER ;
  START : BOOL ;
  PLANCHAS : WORD  := W#16#100;
  ERROR : BOOL ;
  RESET : BOOL ;
END_VAR
VAR_OUTPUT
  ABRIRMCENTRO : BOOL ;
  DESBOBINAR : BOOL ;
  STBY : BOOL ;
END_VAR
VAR
  x31 : BOOL ;
  x32 : BOOL ;
  x33 : BOOL ;
  x34 : BOOL ;
  x30 : BOOL ;
  FP_PRESENCIA : BOOL ;
  BDT : BOOL ;
  FP_START : BOOL ;
  XERROR : BOOL ;
END_VAR
VAR_TEMP
  watchdog_master : BOOL ;
END_VAR
BEGIN
NETWORK
TITLE = Arranque
      SET;
      FP    #BDT;
      S     #x30;
      R     #x31;
      R     #x32;
      R     #x33;
      R     #x34;
NETWORK
TITLE =
      A     #RESET;
      R     #ABRIRMCENTRO;
      R     #DESBOBINAR;
      S     #x30;
      R     #x31;
      R     #x32;
      R     #x33;
      R     #x34;
      R     #XERROR;
NETWORK
TITLE =
      A     #ERROR;
      R     #ABRIRMCENTRO;
      R     #DESBOBINAR;
      R     #x30;
      R     #x31;
      R     #x32;
      R     #x33;
      R     #x34;
      S     #XERROR;
NETWORK
TITLE = x31 a x32
//Comparacion medida centro con medida nominal del centro para pasar de x31 a x32
      A     #x31;
      A(;
      L     #CENTRO;
      L     #MCENTRO;
      ==R;
      );
      R     #x31;
      S     #x32;
NETWORK
TITLE = x32 a x33
//Presencia detecta que la plancha esta en posicion para empezar el proceso de 
//desbobinado-cizallado
      A     #x32;
      A     #PRESENCIA;
      FP    #FP_PRESENCIA;
      R     #x32;
      S     #x33;
NETWORK
TITLE = x33 a x34
//Detecta que la plancha esta lista para ser cizallada
      A     #x33;
      A     #SENSOR;
      R     #x33;
      S     #x34;
NETWORK
TITLE = x34 a x33
//si el contador no ha acabado
      A     #x34;
      T     LD 1;
      TAK;
      T     LD 5;
      L     #Contador;
      T     LW 9;
      L     LD 5;
      L     LD 1;
      A     C [LW 9];
      AN    #SENSOR;
      R     #x34;
      S     #x33;
NETWORK
TITLE = x34 a X30
//si el contador ha cabado
      A     #x34;
      T     LD 1;
      TAK;
      T     LD 5;
      L     #Contador;
      T     LW 9;
      L     LD 5;
      L     LD 1;
      AN    C [LW 9];
      AN    #SENSOR;
      AN    #PRESENCIA;
      R     #x34;
      S     #x30;
NETWORK
TITLE = Tratamiento de bit de fin
      A     #x30;
      =     #STBY;
NETWORK
TITLE = Abrir centro
      A     #x31;
      =     #ABRIRMCENTRO;
NETWORK
TITLE = Carga del contador y desbobinado en x32
      A     #x32;
      S     #DESBOBINAR;
      L     #PLANCHAS;
      T     LD 1;
      TAK;
      T     LD 5;
      L     #Contador;
      T     LW 9;
      L     LD 5;
      L     LD 1;
      S     C [LW 9];
NETWORK
TITLE = Resta del contador y salida del x33
      A     #x33;
      S     #DESBOBINAR;
NETWORK
TITLE = Reset del desbobionado en x34
      A     #x34;
      R     #DESBOBINAR;
NETWORK
TITLE = De X30 a X31
      A     #START;
      FP    #FP_START;
      A     #x30;
      R     #x30;
      S     #x31;
END_FUNCTION_BLOCK

